(* CoDeSys 2.3 library: TcIoFunctions.lib *)
(* Libraries: STANDARD.LIB 5.6.98 17:03:02, TcBase.lib 14.5.09 17:14:08, TcSystem.lib 9.3.10 16:21:30, TcUtilities.lib*24.1.11 11:36:10 *)

(* Global variable list: Globale_Variablen *)
VAR_GLOBAL
END_VAR
VAR_GLOBAL CONSTANT
	ERROR_ASI_COMM_ERROR				:BYTE:=1;
	ERROR_ASI_SLAVEADDRESS				:BYTE:=2;
	ERROR_ASI_SLAVE_NOT_IN_LAS			:BYTE:=11;
	ERROR_ASI_TOGGLE_ERROR				:BYTE:=12;
	EEROR_ASI_DATAEXCHANGE_NOT_SET		:BYTE:=13;

	(* DPV1 via ProfiNET *)
	iMAX_DPV1_SIZE 			: INT := 240;
	iMAX_DPV1_PARAMS 		: INT := 39;

	(* DPV1 via ProfiNET *)
	iMAX_PNET_SIZE 	 		: INT := 32;
	iMAX_PNET_PARAMS 		: INT := 1;

	iMAX_DPV1_SIZE_PNET_REQ	: INT := 260;
	iMAX_DPV1_SIZE_PNET_RES	: INT := 240;

	iMAX_DRIVES_PER_CU		: INT := 15;
	iMAX_FAULTS_PER_DRIVE	: INT := 15;
END_VAR

(* Data type *)
TYPE ControlActiveConfiguration_t :
STRUCT
	HighSwitchCode : BYTE;
	LowSwitchCode : BYTE;
	High1 : BYTE;
	Low1 : BYTE;
	HighDeviceNo : BYTE;
	LowDeviceNo : BYTE;
END_STRUCT
END_TYPE

(* Data type *)
TYPE E_BatteryStatus :
(
	BatteryUnknownStatus, (*The battery status is unknown.*)
	BatteryOk, (*The batteries are OK.*)
	BatteryReplace (*The batteries need to be replaced.*)
);
END_TYPE

(* Data type *)
TYPE E_IOACCESSTYPE :
(
	eIOAccess_Default, 		(* normal memcpy function can be used to copy the data*)
	eIOAccess_Byte,			(* only byte access is allowed,  each byte of the data must be copied individually in a for loop *)
	eIOAccess_WordSwap	(* only aligned word access is allowed. High byte and low byte must be swapped *)
);
END_TYPE

(* Data type *)
TYPE E_PD_Datatype : (
	ePD_UNDEFINED		:=  0,
	ePD_BOOL			:=  1, (* 0/1 (not impl.) *)
	ePD_INT08			:=  2, (* -128 .. 127 *)
	ePD_INT16			:=  3, (* -32768 .. 32767 *)
	ePD_INT32			:=  4, (* -2147483648 .. 2147483647 *)
	ePD_UINT08			:=  5, (* 0 .. 255 *)
	ePD_UINT16			:=  6, (* 0 .. 65535 *)
	ePD_UINT32			:=  7, (* 0 .. 4294967295 *)
	ePD_FLOAT			:=  8, (* IEEE 754 *)
	ePD_VSTRING			:=  9, (* ISO/IEC 646, variable length *)
	ePD_OCTSTRING		:= 10, (* bytearray, variable length *)
	ePD_TIMEOFDAY_WDI	:= 12, (* 6 Bytes:
									4 bytes ms 
									+ 2 bytes day since 1.1.1984 *)
	ePD_TIMEDIFF		:= 13, (* 4|6 Bytes:
									4 bytes ms 
									+ optional 2 bytes days *)
	ePD_N2_16BIT		:= 33,
	ePD_N4_32BIT		:= 34,
	ePD_V2_BITSEQ		:= 35,
	ePD_L2_NIBBLE		:= 36,
	ePD_R2_RECIP_TC		:= 37,
	ePD_T2_TC_16BIT		:= 38,
	ePD_T2_TC_32BIT		:= 39,
	ePD_D2_TC			:= 40,
	ePD_E2_FIXPT_16		:= 41,
	ePD_C2_FIXPT_32		:= 42,
	ePD_X2_NV_16		:= 43,
	ePD_X4_NV_32		:= 44,
	ePD_DATE			:= 50, (* 7 Bytes:
									2 bytes ms
									+ 2 bits (res.), 6 bits (minutes) 
									+ 1 bit (0: StdTime/1: DaylightSavingTime), 2 bits (res.), 5 bits (hours) 
									+ 3 bits (DayOfWeek), 5 bits (DayOfMonth) 
									+ 2 bits (res.), 6 bits (month) 
									+ 1 bit (res.), 7 bits (year) *)
	ePD_TIMEOFDAY_NODI	:= 52, (* 0 .. 268435455 ms *)
	ePD_TIMEDIFF_WDI	:= 53, (* 6 Bytes:
									4 bytes ms 
									+ 2 bytes days *)
	ePD_TIMEDIFF_NODI	:= 54, (* 0 .. 4294967295 ms *)

	ePD_ZERO 			:= 64,
	ePD_BYTE 			:= 65,
	ePD_WORD 			:= 66,
	ePD_DWORD			:= 67,
	ePD_ERROR 			:= 68
);
END_TYPE

(* Data type *)
TYPE E_PD_Dpv1Error : (
	ePD_Err_ParamNumber 			:= 0,
	ePD_Err_ParamReadOnly			:= 1,
	ePD_Err_ValueOutOfRange			:= 2,
	ePD_Err_InvalidSubIndex			:= 3,
	ePD_Err_NoArray					:= 4,
	ePD_Err_WrongDataType			:= 5,
	ePD_Err_OnlyResetPermitted		:= 6,
	ePD_Err_DescNotChangable		:= 7,
	ePD_Err_DescNotFound			:= 9,
	ePD_Err_NoPermissionToChange	:= 11,
	ePD_Err_NoTextArray				:= 15,
	ePD_Err_JobNotExecutable		:= 17,
	ePD_Err_ValueInvalid			:= 20,
	ePD_Err_ResponseToLong			:= 21,
	ePD_Err_ParamAddrInvalid		:= 22,
	ePD_Err_FormatInvalid			:= 23,
	ePD_Err_NumOfValuesInvalid		:= 24,
	ePD_Err_DriveObjNotExisting		:= 25,
	ePD_Err_ParamDeactivated		:= 101,
	ePD_Err_ParamNoWrIfEnabled		:= 107,
	ePD_Err_ParamInvalidUnit		:= 108,
	ePD_Err_ParamNoWrIfNotInitFbk	:= 109,
	ePD_Err_ParamWrIfInitMtr		:= 110,
	ePD_Err_ParamWrIfInitDrv		:= 111,
	ePD_Err_ParamWrIfFastInit		:= 112,
	ePD_Err_ParamWrIfReady			:= 113,
	ePD_Err_ParamWrIfInitParamReset	:= 114,
	ePD_Err_ParamWrIfInitSafety		:= 115,
	ePD_Err_ParamWrIfInitTechApp	:= 116,
	ePD_Err_ParamWrIfInit			:= 117,
	ePD_Err_ParamWrIfInitDwnLd		:= 118,
	ePD_Err_ParamNoWrtIfDwnLd		:= 119,
	ePD_Err_ParamWrIfInitDrvCfg		:= 120,
	ePD_Err_ParamWrIfInitSetDrvType	:= 121,
	ePD_Err_ParamWrIfInitDatasetCfg	:= 122,
	ePD_Err_ParamWrIfInitDevCfg		:= 123,
	ePD_Err_ParamWrIfInitDevDwnLd	:= 124,
	ePD_Err_ParamWrIfInitDevPrmReset:= 125,
	ePD_Err_ParamWrIfInitDevReady	:= 126,
	ePD_Err_ParamWrIfInitDevice		:= 127,
	ePD_Err_ParamNoWriteIfDwnLd		:= 129,
	ePD_Err_CtrlTakeOverBlocked		:= 130,
	ePD_Err_ParamBicoSetInvalid		:= 131,
	ePD_Err_ParamChangeBlocked		:= 132,
	ePD_Err_ParamNoAccessDefined	:= 133,
	ePD_Err_BelowDefinedMinimum		:= 200,
	ePD_Err_AboveDefinedMaximum		:= 201,
	ePD_Err_WriteNotPermitted		:= 204
);
END_TYPE

(* Data type *)
TYPE E_PD_DriveType : (
	ePD_DRVTYPE_UNKNOWN 	:= 0,
	ePD_SINAMICS_S 			:= 1,
	ePD_SINAMICS_G 			:= 2,
	ePD_SINAMICS_I 			:= 3,
	ePD_SINAMICS_CX32 		:= 4,
	ePD_SINAMICS_GM 		:= 5,
	ePD_SINAMICS_GL 		:= 7,
	ePD_ACTLINEMOD 			:= 10,
	ePD_SERVO 				:= 11,
	ePD_VECTOR 				:= 12,
	ePD_VECTOR_VM 			:= 13,
	ePD_VECTOR_GL 			:= 14,
	ePD_SMARTLINEMOD 		:= 20,
	ePD_BASICLINEMOD 		:= 30,
	ePD_ACTIVELINEMOD_MV 	:= 40,
	ePD_BASICLINEMOD_MV 	:= 41,
	ePD_TB30 				:= 100,
	ePD_DMC 				:= 150,
	ePD_TM31 				:= 200,
	ePD_TM41 				:= 201,
	ePD_TM17_HIGHFEATURE 	:= 202,
	ePD_TM15 				:= 203,
	ePD_TM15_SINAMICS 		:= 204,
	ePD_CU_LINK 			:= 254
);
END_TYPE

(* Data type *)
TYPE E_PD_SaveType : (
	E_PD_SaveInactive 			:= 0,
	E_PD_SaveNonVolatilePWRON	:= 1,
	E_PD_SaveNonVolatileP967_10	:= 10,
	E_PD_SaveNonVolatileP967_11	:= 11,
	E_PD_SaveNonVolatileP967_12	:= 12,
	E_PD_SaveNonVolatile_20		:= 20,
	E_PD_SaveNonVolatile_21		:= 21,
	E_PD_SaveNonVolatile_22		:= 22,
	E_PD_SaveNonVolatile_23		:= 23,
	E_PD_SaveNonVolatile_24		:= 24,
	E_PD_SaveNonVolatile_25		:= 25,
	E_PD_SaveNonVolatile_26		:= 26,
	E_PD_SaveVolatileP967_1011	:= 1011,
	E_PD_SaveVolatileP967_1012	:= 1012,
	E_PD_SaveVolatileP967_1013	:= 1013
);
END_TYPE

(* Data type *)
TYPE E_PD_State : (
	ePD_IDLE 			:= 0,
	ePD_InitialRead 	:= 1,
	ePD_InitialWrite 	:= 2,
	ePD_ReadParam 		:= 3,
	ePD_WriteParam 		:= 4,
	ePD_ReadDiagInfo 	:= 5,
	ePD_QuitErrorCU 	:= 6,
	ePD_ResetDrive 		:= 7,
	ePD_SaveParamCU 	:= 8,
	ePD_SaveParamDrive 	:= 9,
	ePD_ClearErrorCU 	:= 10,
	ePD_ClearErrorDrive	:= 11,
	ePD_QuitErrorDrive 	:= 12
);
END_TYPE

(* Data type *)
TYPE E_SercosAttribLen : (
	eLEN_2BYTE	:= 1,
	eLEN_4BYTE	:= 2,
	eLEN_8BYTE	:= 3,
	eLEN_V1BYTE	:= 4,
	eLEN_V2BYTE	:= 5,
	eLEN_V4BYTE	:= 6,
	eLEN_V8BYTE	:= 7
);
END_TYPE

(* Data type *)
TYPE E_SercosAttribType : (
	eType_BIN		:= 0,
	eType_UNSIGNED	:= 1,
	eType_SIGNED	:= 2,
	eType_HEX		:= 3,
	eType_ASCII		:= 4,
	eType_ID		:= 5,
	eType_FLOAT		:= 6
);
END_TYPE

(* Data type *)
TYPE E_SercosBackupState  : (
	eBkup_IDLE 						:=  0,
	eBkup_READ_IDNLIST_INI 			:=  1,
	eBkup_READ_IDNLIST_ACT 			:=  2,
	eBkup_FILEOPEN					:=  3,
	eBkup_FILECLOSE					:=  4,
	eBkup_CHECK_CRC_ACT 			:=  5,
	eBkup_UPDT_CRC_INI				:=  6,
	eBkup_UPDT_CRC_ACT 				:=  7,

	eBkup_BACKUP_WRITE_FILEHEADER 	:= 10,
	eBkup_BACKUP_PARAM_INI 			:= 11,
	eBkup_BACKUP_PARAM_ACT 			:= 12,
	eBkup_BACKUP_WRITE_HEADER 		:= 14,
	eBkup_BACKUP_WRITE_DATA 		:= 15,

	eBkup_RESTORE_READ_FILEHEADER 	:= 20,
	eBkup_RESTORE_READ_HEADER		:= 21,
	eBkup_RESTORE_READ_DATA 		:= 22,
	eBkup_RESTORE_PARAM_INI			:= 23,
	eBkup_RESTORE_PARAM_ACT			:= 24
);
END_TYPE

(* Data type *)
TYPE E_SercosParamDataType : (
	eDT_LIST	:= 0,
	eDT_INT,
	eDT_UINT,
	eDT_WORD,
	eDT_DINT,
	eDT_UDINT,
	eDT_DWORD,
	eDT_REAL,
	eDT_LREAL
);
END_TYPE

(* Data type *)
TYPE E_UpsCommStatus :
(
	UpsCommUnknownStatus,
	UpsCommOk, (*The communication path to the UPS is OK.*)
	UpsCommFailed (*The communication path to the UPS has failed.*)
);
END_TYPE

(* Data type *)
TYPE E_UpsPowerStatus :
(
	PowerUnknownStatus, (*The status of power is unknown.*)
	PowerOnLine, (* Power is OK.*)
	PowerOnBattery (*A power failure has occurred.*)
);
END_TYPE

(* Data type *)
TYPE FC310X_DIAG_DATA :
STRUCT
	ReceiveErrorCounter: WORD;
	RepeatCounter: ARRAY[0..8] OF WORD;
	NoAnswerCounter: DWORD;
	LastDpv1Error: ARRAY[0..3] OF BYTE;
	Reserved: ARRAY[0..3] OF BYTE;
	DP_Diag_Stationstatus_1: BYTE;
	DP_Diag_Stationstatus_2: BYTE;
	DP_Diag_Stationstatus_3: BYTE;
	DP_Diag_MasterAdd: BYTE;
	DP_Diag_IdentNumberHi: BYTE;
	DP_Diag_IdentNumberLo: BYTE;
	DP_Diag_ExtDiagData: ARRAY[0..237] OF BYTE;
END_STRUCT
END_TYPE

(* Data type *)
TYPE FC510X_DIAG_DATA :
STRUCT
	flags: WORD;
	pdoReceived:WORD;
	pdoFault: WORD;
	startUpFault: BYTE;
	sdoFault: BYTE;
	index: WORD;
	subindex: BYTE;
	dummy2: BYTE;
	errorClass: BYTE;
	errorCode: BYTE;
	additionalCode: WORD;
	readValue: DWORD;
	expectedValue: DWORD;
	noOfEmergencies: WORD;
	emergency: ARRAY[0..9,0..7] OF BYTE;
END_STRUCT
END_TYPE

(* Data type *)
TYPE GetErrorInfo_t :
STRUCT
	HighResult : BYTE;
	LowResult : BYTE;
	HighEntryCount : BYTE;
	LowEntryCount : BYTE;
	HighErrorCode : BYTE;
	LowErrorCode : BYTE;
	HighAddErrInfo : BYTE;
	LowAddErrInfo : BYTE;
END_STRUCT
END_TYPE

(* Data type *)
TYPE HLword_t :
STRUCT
	High : BYTE;
	Low : BYTE;
END_STRUCT
END_TYPE

(* Data type *)
TYPE IODEVICETYPES :
(
	IODEVICETYPE_UNKNOWN			:= 0,
	IODEVICETYPE_C1220				:= 1,			(* Beckhoff Lightbus-Master*)
	IODEVICETYPE_C1200				:= 2,			(* Beckhoff Lightbus-Master*)
	IODEVICETYPE_SPC3				:= 3,			(* ProfiBus Slave (Siemens)*)
	IODEVICETYPE_CIF30DPM			:= 4,			(* ISA ProfiBus-Master 2 kByte (Hilscher)*)
	IODEVICETYPE_CIF40IBSM			:= 5,			(* ISA Interbus-S-Master 2 kByte (Hilscher)*)
	IODEVICETYPE_BKHFPC			:= 6,			(* Beckhoff PC C2001*)
	IODEVICETYPE_CP5412A2			:= 7,			(* ProfiBus-Master (Siemens)*)
	IODEVICETYPE_SERCANSISA		:= 8,			(* Sercos Master (Indramat)*)
	IODEVICETYPE_LPTPORT			:= 9,			(* Lpt Port*)
	IODEVICETYPE_DPRAM				:= 10,		(* Generic DPRAM*)
	IODEVICETYPE_COMPORT			:= 11,		(* COM Port*)
	IODEVICETYPE_CIF30CAN			:= 12,		(* ISA CANopen-Master (Hilscher)*)
	IODEVICETYPE_CIF30PB			:= 13,		(* ISA ProfiBus-Master 8 kByte (Hilscher)*)
	IODEVICETYPE_BKHFCP2030		:= 14,		(* Beckhoff CP2030 (Pannel-Link)*)
	IODEVICETYPE_IBSSCIT				:= 15,		(* ISA Interbus-S-Master (Phoenix)*)
	IODEVICETYPE_CIF30IBM			:= 16,		(* ISA Interbus-S-Master (Hilscher)*)
	IODEVICETYPE_CIF30DNM			:= 17,		(* ISA DeviceNet-Master (Hilscher)*)
	IODEVICETYPE_FCXXXX				:= 18,		(* Beckhoff-Filedbus card *)
	IODEVICETYPE_CIF50PB			:= 19,		(* PCI ProfiBus-Master 8 kByte (Hilscher)*)
	IODEVICETYPE_CIF50IBM			:= 20,		(* PCI Interbus-S-Master (Hilscher)*)
	IODEVICETYPE_CIF50DNM			:= 21,		(* PCI DeviceNet-Master (Hilscher)*)
	IODEVICETYPE_CIF50CAN			:= 22,		(* PCI CANopen-Master (Hilscher)*)
	IODEVICETYPE_CIF60PB			:= 23,		(* PCMCIA ProfiBus-Master (Hilscher)*)
	IODEVICETYPE_CIF60DNM			:= 24,		(* PCMCIA DeviceNet-Master (Hilscher)*)
	IODEVICETYPE_CIF60CAN			:= 25,		(* PCMCIA CANopen-Master (Hilscher)*)
	IODEVICETYPE_CIF104DP			:= 26,		(* PC104 ProfiBus-Master 2 kByte (Hilscher)*)
	IODEVICETYPE_C104PB				:= 27,		(* PC104 ProfiBus-Master 8 kByte (Hilscher)*)
	IODEVICETYPE_C104IBM			:= 28,		(* PC104 Interbus-S-Master 2 kByte (Hilscher)*)
	IODEVICETYPE_C104CAN			:= 29,		(* PC104 CANopen-Master (Hilscher)*)
	IODEVICETYPE_C104DNM			:= 30,		(* PC104 DeviceNet-Master (Hilscher)*)
	IODEVICETYPE_BKHFCP9030		:= 31,		(* Beckhoff CP9030 (Pannel-Link with UPS)*)
	IODEVICETYPE_SMB					:= 32,		(* Motherboard System Management Bus*)
	IODEVICETYPE_PBMON				:= 33,		(* Beckhoff-PROFIBUS-Monitor*)
	IODEVICETYPE_CP5613				:= 34,		(* PCI ProfiBus-Master (Siemens)*)
	IODEVICETYPE_CIF60IBM			:= 35,		(* PCMCIA Interbus-S-Master (Hilscher)*)
	IODEVICETYPE_FC200X				:= 36,		(* Beckhoff-Lightbus-I/II-PCI-Karte*)
	IODEVICETYPE_FC3100_OLD		:= 37,		(* obsolete: dont use*)
	IODEVICETYPE_FC3100				:= 38,		(* Beckhoff-Profibus-PCI*)
	IODEVICETYPE_FC5100				:= 39,		(* Beckhoff-CanOpen-PCI*)
	IODEVICETYPE_FC5200				:= 41,		(* Beckhoff-DeviceNet-PCI*)

	IODEVICETYPE_BKHFNCBP			:= 43,		(* Beckhoff NC back plane*)
	IODEVICETYPE_SERCANSPCI		:= 44,		(* Sercos Master (SICAN/IAM PCI)*)
	IODEVICETYPE_ETHERNET			:= 45,		(* Virtual Ethernet Device*)
	IODEVICETYPE_SERCONPCI		:= 46,		(* Sercon 410B or 816 Chip Master or Slave (PCI)*)
	IODEVICETYPE_IBSSCRIRTLK		:= 47,		(* ISA Interbus-S-Master with Slave-Module LWL Basis (Phoenix)*)
	IODEVICETYPE_FC7500				:= 48,		(* Beckhoff-SERCOS-PCI*)
	IODEVICETYPE_CIF30IBS			:= 49,		(* ISA Interbus-S-Slave (Hilscher)*)
	IODEVICETYPE_CIF50IBS			:= 50,		(* PCI Interbus-S-Slave (Hilscher)*)
	IODEVICETYPE_C104IBS			:= 51,		(* PC104 Interbus-S-Slave (Hilscher)*)
	IODEVICETYPE_BKHFCP9040		:= 52,		(* Beckhoff CP9040 (CP-PC) *)
	IODEVICETYPE_BKHFAH2000		:= 53,		(* Beckhoff AH2000 (Hydr. Backplane) *)
	IODEVICETYPE_BKHFCP9035		:= 54,		(* Beckhoff CP9035 (PCI, Pannel-Link with UPS) *)
	IODEVICETYPE_AH2000MC			:= 55,		(* Beckhoff-AH2000 with Profibus-MC *)
	IODEVICETYPE_FC3100MON		:= 56,		(* Beckhoff-Profibus-Monitor-PCI *)
	IODEVICETYPE_USB					:= 57,		(* Virtual USB Device *)
	IODEVICETYPE_FC5100MON		:= 58,		(* Beckhoff-CANopen-Monitor-PCI *)
	IODEVICETYPE_FC5200MON		:= 59,		(* Beckhoff-DeviceNet-Monitor-PCI *)
	IODEVICETYPE_FC3100SLV			:= 60,		(* Beckhoff-Profibus-PCI Slave *)
	IODEVICETYPE_FC5100SLV			:= 61,		(* Beckhoff-CanOpen-PCI Slave *)
	IODEVICETYPE_FC5200SLV			:= 62,		(* Beckhoff-DeviceNet-PCI Slave *)
	IODEVICETYPE_IBSSCITPCI			:= 63,		(* PCI Interbus-S-Master (Phoenix) *)
	IODEVICETYPE_IBSSCRIRTLKPCI	:= 64,		(* PCI Interbus-S-Master with slave module  LWL Basis (Phoenix) *)
	(* 11 November 2002 *)
	IODEVICETYPE_CX1100_BK		:= 65,		(* Beckhoff-CX1100 terminal bus power supply *)
	IODEVICETYPE_ENETRTMP			:= 66,		(* Ethernet real time miniport *)
	IODEVICETYPE_CX1500_M200		:= 67,		(* PC104 Lightbus-Master *)
	IODEVICETYPE_CX1500_B200		:= 68,		(* PC104 Lightbus-Slave *)
	IODEVICETYPE_CX1500_M310		:= 69,		(* PC104 ProfiBus-Master *)
	IODEVICETYPE_CX1500_B310		:= 70,		(* PC104 ProfiBus-Slave *)
	IODEVICETYPE_CX1500_M510		:= 71,		(* PC104 CANopen-Master *)
	IODEVICETYPE_CX1500_B510		:= 72,		(* PC104 CANopen-Slave *)
	IODEVICETYPE_CX1500_M520		:= 73,		(* PC104 DeviceNet-Master *)
	IODEVICETYPE_CX1500_B520		:= 74,		(* PC104 DeviceNet-Slave *)
	IODEVICETYPE_CX1500_M750		:= 75,		(* PC104 Sercos-Master *)
	IODEVICETYPE_CX1500_B750		:= 76,		(* PC104 Sercos-Slave *)
	IODEVICETYPE_BX_BK				:= 77,		(* BX terminal bus interface *)
	IODEVICETYPE_BX_M510			:= 78,		(* BX SSB-Master *)
	IODEVICETYPE_BX_B310			:= 79,		(* BX ProfiBus-Slave *)
	(* 29 August 2005 *)
	IODEVICETYPE_IBSSCRIRTPCI		:= 80,		(* PCI Interbus-S-Master with slave module copper basis (Phoenix) *)
	IODEVICETYPE_BX_B510			:= 81,		(* BX CANopen Slave *)
	IODEVICETYPE_BX_B520			:= 82,		(* BX DeviceNet Slave *)
	IODEVICETYPE_BC3150				:= 83,		(* BCxx50 ProfiBus Slave *)
	IODEVICETYPE_BC5150				:= 84,		(* BCxx50 CANopen Slave *)
	IODEVICETYPE_BC5250				:= 85,		(* BCxx50 DeviceNet Slave *)
	IODEVICETYPE_EL6731				:= 86,		(* Beckhoff Profibus-EtherCAT Terminal *)
	IODEVICETYPE_EL6751				:= 87,		(* Beckhoff CanOpen-EtherCAT Terminal *)
	IODEVICETYPE_EL6752				:= 88,		(* Beckhoff DeviceNet-EtherCAT Terminal *)
	IODEVICETYPE_COMPB				:= 89,		(* COM ProfiBus Master 8 kByte (Hilscher) *)
	IODEVICETYPE_COMIBM			:= 90,		(* COM Interbus-S Master (Hilscher) *)
	IODEVICETYPE_COMDNM			:= 91,		(* COM DeviceNet Master (Hilscher) *)
	IODEVICETYPE_COMCAN			:= 92,		(* COM CANopen Master (Hilscher) *)
	IODEVICETYPE_COMIBS				:= 93,		(* COM CANopen Slave (Hilscher) *)
	IODEVICETYPE_ETHERCAT			:= 94,		(* EtherCAT in direct mode *)
	IODEVICETYPE_PROFINETIOCONTROLLER := 95,	(* PROFINET Master *)
	IODEVICETYPE_PROFINETIODEVICE := 96,		(* PROFINET Slave *)
	IODEVICETYPE_EL6731SLV			:= 97,		(* Beckhoff Profibus Slave EtherCAT Terminal *)
	IODEVICETYPE_EL6751SLV			:= 98,		(* Beckhoff CanOpen Slave EtherCAT Terminal *)
	IODEVICETYPE_EL6752SLV			:= 99,		(* Beckhoff DeviceNet Slave EtherCAT Terminal *)
	IODEVICETYPE_C104PPB			:= 100,		(* PC104+ ProfiBus Master 8 kByte (Hilscher) *)
	IODEVICETYPE_C104PCAN			:= 101,		(* PC104+ CANopen Master (Hilscher) *)
	IODEVICETYPE_C104PDNM			:= 102,		(* PC104+ DeviceNet Master (Hilscher) *)
	IODEVICETYPE_BC8150				:= 103,		(* BCxx50 Serial Slave *)
	IODEVICETYPE_BX9000				:= 104,		(* BX9000 Ethernet Slave *)
	(* 27 April 2009 *)
	IODEVICETYPE_CX9000_BK		:= 105,	(* Beckhoff-CX9000 K-Bus Power Supply *)
	IODEVICETYPE_EL6601				:= 106,	(* Beckhoff-RT-Ethernet-EtherCAT-Terminal *)
	IODEVICETYPE_BC9050				:= 107,	(* BC9050 Ethernet Slave *)
	IODEVICETYPE_BC9120				:= 108,	(* BC9120 Ethernet Slave *)
	IODEVICETYPE_ENETADAPTER	:= 109,	(* Ethernet Miniport Adapter *)
	IODEVICETYPE_BC9020				:= 110,	(* BC9020 Ethernet Slave *)
	IODEVICETYPE_ETHERCATPROT	:= 111,	(* EtherCAT Protocol in direct mode *)
	IODEVICETYPE_ETHERNETNVPROT	:= 112,	(* *)
	IODEVICETYPE_ETHERNETPNMPROT	:= 113,	(* *)
	IODEVICETYPE_EL6720				:= 114,	(* Beckhoff-Lightbus-EtherCAT-Terminal *)
	IODEVICETYPE_ETHERNETPNSPROT	:= 115,	(* *)
	IODEVICETYPE_BKHFCP6608		:= 116,	(*	Beckhoff CP6608(IXP PC) *)
	IODEVICETYPE_PTP_IEEE1588		:= 117,  (* *)
	IODEVICETYPE_EL6631SLV			:= 118,	(* EL6631-0010 Profinet Slave terminal *)
	IODEVICETYPE_EL6631				:= 119,	(* EL6631 Profinet Master terminal *)
	IODEVICETYPE_CX5000_BK		:= 120,	(* Beckhoff-CX5100 K-Bus power supply *)
	IODEVICETYPE_PCIDEVICE			:= 121,	(* Generic PCI DPRAM (TCOM) *)
	IODEVICETYPE_ETHERNETUPDPROT 	:= 122,	(* UDP Protocol *)
	(* 13 August 2010 *)
	IODEVICETYPE_ETHERNETAUTOPROT := 123,	(* Automation Protocol *)
	IODEVICETYPE_CCAT				:= 124,	(* CCAT *)
	IODEVICETYPE_CPLINK3			:= 125,	(* Virtuelles USB Device (remote via CPLINK3) *)
	IODEVICETYPE_EL6632				:= 126,	(* EL6632 *)
	IODEVICETYPE_CCAT_PBM			:= 127,	(* CCAT Profibus Master *)
	IODEVICETYPE_CCAT_PBS			:= 128,	(* CCAT Profibus Slave *)
	IODEVICETYPE_CCAT_CNM			:= 129,	(* CCAT CANopen Master *)
	IODEVICETYPE_ETHERCATSLAVE	:= 130,	(* EtherCAT Slave *)
	IODEVICETYPE_BACNET			:= 131,	(* BACnet device *)
	IODEVICETYPE_CCAT_CNS			:= 132,	(* CCAT CANopen Slave *)
	IODEVICETYPE_ETHIP_SCANNER	:= 133,  (* ETHERNET IP  Master *)
	IODEVICETYPE_ETHIP_ADAPTER	:= 134,  (* ETHERNET IP  Slave *)

	(* reserved for new devices*)

	IODEVICETYPE_MAX							(**)
);
END_TYPE

(* Data type *)
TYPE ReadResult_t :
STRUCT
	High1 : BYTE;
	Low1 : BYTE;
	High2 : BYTE;
	Low2 : BYTE;
END_STRUCT
END_TYPE

(* Data type *)
TYPE ST_AdsTecSysData :
STRUCT
	bShiftKey		: BOOL; 	(* TRUE == Shift key pressed*)
	bRMouseKey		: BOOL; 	(* TRUE == Right mouse key pressed *)
	bHotKey			: BOOL;	(* TRUE == Hotkey pressed *)
	bTaskChaKey	: BOOL;	(* TRUE == Task change key pressed *)
	bABCKey		: BOOL;	(* TRUE == ABC soft keyboard key pressed*)
	bRsrv1			: BOOL;
	bRsrv2			: BOOL;
	bRsrv3			: BOOL;

	bMainFanErr		: BOOL; 	(* TRUE == Main fan error*)
	bCpuFanErr		: BOOL;	(* TRUE == CPU fan error*)
	bTempErr		: BOOL;	(* TRUE == Internal temperature error ( temp > 50°C)*)
	bBatteryErr		: BOOL;	(* TRUE == Battery error *)
	bRsrv4			: BOOL;
	bRsrv5			: BOOL;
	bRsrv6			: BOOL;
	bRsrv7			: BOOL;

	nMainNtcTemp	: SINT; 	(* Main NTC temperature (-127°C .. + 127°C) *)
	nExtNtcTemp		: SINT;	(* External NTC temperature (-127°C .. + 127°C) *)

	nRsrv8			: ARRAY[1..12] OF BYTE;
END_STRUCT
END_TYPE

(* Data type *)
TYPE ST_Dpv1Header :
STRUCT
	(* header *)
	iRequestRef 	: USINT;	(* 1..255;    0: reserved *)
	iRequestID 		: SINT;		(* 1: Read;   2: Write;     0x40..0x7F: manufacturer specific;   else: reserved *)
	iAxis			: USINT;	(* 0..255 *)
	iNumOfParams	: USINT;	(* 1..39;     else: reserved *)
END_STRUCT
END_TYPE

(* Data type *)
TYPE ST_Dpv1ParamAddr :
STRUCT
	(* parameter *)
	iAttribute			: USINT;	(* 0x10: Value;   0x20: Description;   0x30: Text (not impl.);   0x80..F0: manufaturer specific (not impl.);   else: reserved *)
	iNumOfElements		: USINT;	(* 1..117: number of array elements;    0: Special Function;   else: reserved *)
	iParameterNumber	: UINT;		(* 1..65535: parameter number;    0: reserved *)
	iSubIndex			: UINT;		(* 0..65535: subindex *)
END_STRUCT
END_TYPE

(* Data type *)
TYPE ST_Dpv1ParamAddrEx :
STRUCT
	(* parameter *)
	iAttribute			: USINT;	(* 0x10: Value;   0x20: Description;   0x30: Text;   0x80..F0: manufaturer specific;   else: reserved *)
	iNumOfElements		: USINT;	(* 1..234: number of elements;    0: Special Function;   else: reserved *)
	iParameterNumber	: UINT;		(* 1..65535: parameter number;    0: reserved *)
	iSubIndex			: UINT;		(* 0..65535: subindex *)
	iDataAddr			: UDINT;	(* address of buffer/address of plc variable *)
	iDataSize			: UDINT;	(* size of buffer/size of plc variable *)
	eFormat				: E_PD_Datatype;	(* 0x01..0x36: datatype;   0x40: ZERO;   0x41: BYTE;   0x42: WORD;   0x43: DWORD;   0x44: Error;   else reserved *)
	iNumOfValues		: UINT;		(* 0..234: number of values;   else: reserved *)
	iErrorValue			: UDINT;	(* DPV1 error value *)
	stError				: ST_PD_Dpv1Error; (* DPV1 error flag, DPV1 error enum *)
END_STRUCT
END_TYPE

(* Data type *)
TYPE ST_Dpv1ValueHeader :
STRUCT
	iFormat			: USINT;	(* 0x01..0x36: datatype;   0x40: ZERO;   0x41: BYTE;   0x42: WORD;   0x43: DWORD;   0x44: Error;   else reserved *)
	iNumOfValues	: USINT;	(* 0..234: number of values;   else: reserved *)
END_STRUCT
END_TYPE

(* Data type *)
TYPE ST_Dpv1ValueHeaderEx :
STRUCT
	eFormat			: E_PD_Datatype;	(* 0x01..0x36: datatype;   0x40: ZERO;   0x41: BYTE;   0x42: WORD;   0x43: DWORD;   0x44: Error;   else reserved *)
	iNumOfValues	: USINT;	(* 0..234: number of values;   else: reserved *)
	iOffset			: USINT;	(* Offset in the DPV1 response telegram *)
	iDataLen		: UINT;		(* data lenght *)
	strData			: STRING;	(* printed data *)
END_STRUCT
END_TYPE

(* Data type *)
TYPE ST_NovRamAddrInfo :
STRUCT
	pCardAddress	:	UDINT;
	iCardMemSize	:	UDINT;
END_STRUCT
END_TYPE

(* Data type *)
TYPE ST_NovRamAddrInfoEx :
STRUCT
	pCardAddress	:	UDINT;
	iCardMemSize	:	UDINT;
	eAccessType	:	E_IOACCESSTYPE;
END_STRUCT
END_TYPE

(* Data type *)
TYPE ST_Parameter_IN :
STRUCT
	iParameterStatus			:WORD;
	iParameterReadValue		:DWORD;

(*ParameterStatus
Byte-Offset	Bit-Offset		Bedeutung
	0			0-5		Status-Bits (wie bei bisherigen Klemmen)
	0			6		0: keine Diagnose, 1: Diagnose (wie bei bisherigen Klemmen)
	0			7		immer 0: keine Registerkommunikation
	1			0-3		Reserviert für Erweiterungen
	1			4		Toggle-Bit, um Auftrag zu quittieren (bei Cyclic wird das Bit 6 aus Byte 0 kopiert)
	1			5		Quittung (0: NoError, 1: Error)
	1			6		0: Cyclic, 1: Acyclic
	1			7		0: Parameterzugriff, 1: ADS
	2					Input-Daten (Cyclic), Parameterwert (Acyclic) oder Fehlernummer Bit 0-7
	3					Input-Daten (Cyclic), Parameterwert (Acyclic) oder Fehlernummer Bit 8-15
	4					Input-Daten (Cyclic), Parameterwert (Acyclic) oder Fehlernummer Bit 16-23
	5					Input-Daten (Cyclic), Parameterwert (Acyclic) oder Fehlernummer Bit 24-31

*)
END_STRUCT
END_TYPE

(* Data type *)
TYPE ST_Parameter_OUT :
STRUCT
	ParameterControl			:WORD;
	iParametervalue			:DWORD;

(*ParameterControl
Byte-Offset	Bit-Offset		Bedeutung
	0			0-5		Parameternummer Bit 0-5 (oder Parameter-Offset)
	0			6		Bei Acyclic: 0: Read, 1:Write, bei Cyclic (immer Read/Write) wird das Bit in die Inputdaten kopiert, um eine direkte Zuordnung zu haben (dann könnten die Cyclic-Daten auch geändert werden)
	0			7		0: Parameterzugriff, 1: Registerkommunikation
	1			0-5		Parameternummer Bit 6-11 (oder Parameter-Page)
	1			6		0: Cyclic, 1: Acyclic
	1			7		0: Parameterzugriff, 1: ADS
	2					Output-Daten (Cyclic) oder Parameterwert (Acyclic) Bit 0-7
	3					Output-Daten (Cyclic) oder Parameterwert (Acyclic) Bit 8-15
	4					Output-Daten (Cyclic) oder Parameterwert (Acyclic) Bit 16-23
	5					Output-Daten (Cyclic) oder Parameterwert (Acyclic) Bit 24-31

*)

END_STRUCT
END_TYPE

(* Data type *)
TYPE ST_ParameterBuffer :
STRUCT
	ParameterControl			:ARRAY[0..50] OF WORD;
	iParametervalue			:ARRAY[0..50] OF DWORD;
	iParameterStatus			:ARRAY[0..50] OF WORD;
	iParameterReadValue		:ARRAY[0..50] OF DWORD;
	icounterState				:INT;
	icounterControl			:INT;
END_STRUCT
END_TYPE

(* Data type *)
TYPE ST_PD_CUDriveInfo :
STRUCT
	iNumOfDriveObjects	: UINT;
	iReserved	: UINT;
	iIndex		: ARRAY [0..iMAX_DRIVES_PER_CU] OF UINT;			(* [0] is ControlUnit, [1..15] for the drives *)
	eType		: ARRAY [0..iMAX_DRIVES_PER_CU] OF E_PD_DriveType;	(* [0] is ControlUnit, [1..15] for the drives *)
	iFWVersion	: ARRAY [0..iMAX_DRIVES_PER_CU] OF UDINT;			(* [0] is ControlUnit, [1..15] for the drives *)
	iFWDateYear	: ARRAY [0..iMAX_DRIVES_PER_CU] OF UINT;			(* [0] is ControlUnit, [1..15] for the drives *)
	iFWDateDM	: ARRAY [0..iMAX_DRIVES_PER_CU] OF UINT;			(* [0] is ControlUnit, [1..15] for the drives *)
	iPbTelType	: ARRAY [0..iMAX_DRIVES_PER_CU] OF UINT;			(* [0] is ControlUnit, [1..15] for the drives *)
END_STRUCT
END_TYPE

(* Data type *)
TYPE ST_PD_DOIdentification :
STRUCT
	iCompany				: UINT;				(* 42 = Siemens *)
	eType					: E_PD_DriveType;	(* drive object type, e.g. ePD_SINAMICS_S, ePD_SERVO, ... *)
	iFWVersion				: UINT;				(* 102 --> v01.02, hotfix see below *)
	iFWDateYear				: UINT;				(* 2003 --> year 2003 *)
	iFWDateDayMonth			: UINT;				(* 1401 --> 14.01. *)
	iProfiDrvTypeClass		: UINT;
	iProfiDrvSubTypeClass	: UINT;
	iReserved				: ARRAY [7..9] OF UINT;
	iFWVersionPatchVersion	: UINT;				(* 600 --> FW v01.02.06.00, hotfix see below *)
END_STRUCT
END_TYPE

(* Data type *)
TYPE ST_PD_Dpv1Error :
STRUCT
	bError		: BOOL;
	eErrorId	: E_PD_Dpv1Error;
END_STRUCT
END_TYPE

(* Data type *)
TYPE ST_PD_DriveDiag :
STRUCT
	iNumOfFaultsTotal		: UINT;
	iNumOfFaultsSinceReset	: UINT;
	iNumOfWarnsTotal		: UINT;
	iStateWordErrorWarning	: UINT;
	iErrorCode	: ARRAY [0..iMAX_FAULTS_PER_DRIVE] OF UINT;			(* [0] is ControlUnit, [1..15] for the drives *)
	iErrorArgI	: ARRAY [0..iMAX_FAULTS_PER_DRIVE] OF UDINT;		(* [0] is ControlUnit, [1..15] for the drives *)
	fErrorArgF	: ARRAY [0..iMAX_FAULTS_PER_DRIVE] OF REAL;			(* [0] is ControlUnit, [1..15] for the drives *)
	iWarnCode	: ARRAY [0..iMAX_FAULTS_PER_DRIVE] OF UINT;			(* [0] is ControlUnit, [1..15] for the drives *)
	iWarnArgI	: ARRAY [0..iMAX_FAULTS_PER_DRIVE] OF UDINT;		(* [0] is ControlUnit, [1..15] for the drives *)
	fWarnArgF	: ARRAY [0..iMAX_FAULTS_PER_DRIVE] OF REAL;			(* [0] is ControlUnit, [1..15] for the drives *)
END_STRUCT
END_TYPE

(* Data type *)
TYPE ST_PNET_CCDSTS :
STRUCT
	iCycleCounter	: UINT;
	iDataState		: USINT;
	iTransferState	: USINT;
END_STRUCT
END_TYPE

(* Data type *)
TYPE ST_PNIOConfigRecord :
STRUCT
	iRW				: UINT; (* 0: Read, 1: Write *)
	iNumOfAR		: UINT;
	iAPI			: UDINT;
	iSlot			: UINT;
	iSubSlot		: UINT;
	stPNIORecord	: ST_PNIORecord;
END_STRUCT
END_TYPE

(* Data type *)
TYPE ST_PNIORecord :
STRUCT
	iIndex 		: UINT;
	iLength 	: UINT; (* 0 for READ *)
	iTransfSeq	: UINT;
	iAligned 	: UINT;
END_STRUCT
END_TYPE

(* Data type *)
TYPE ST_PNIOState :
STRUCT
	bInDataExchange	: BOOL; (* bit 0 *)
	bApplRunning	: BOOL; (* bit 2 *)
	bDiagIndicator	: BOOL; (* bit 3 *)
END_STRUCT
END_TYPE

(* Data type *)
TYPE ST_PZD_IN :
STRUCT
	wSTW		:WORD;
	wHIW		:WORD;
	PZD3		:WORD;
	PZD4		:WORD;
	PZD5		:WORD;
	PZD6		:WORD;

END_STRUCT
END_TYPE

(* Data type *)
TYPE ST_PZD_OUT :
STRUCT
	wCtrlW			:WORD;
	PZD2			:WORD;
	PZD3			:WORD;
	PZD4			:WORD;
	PZD5			:WORD;
	PZD6			:WORD;
END_STRUCT
END_TYPE

(* Data type *)
TYPE ST_SercosFileHeader :
STRUCT
	nVersion	 : UDINT;
	nListType	 : UDINT;
	cbCommentLen : UDINT;
	sComment	 : T_MaxString;
END_STRUCT
END_TYPE

(* Data type *)
TYPE ST_SercosParamAttrib :
STRUCT
	nFactor			: UINT;					(* bits  0..15 *)
	eLength			: E_SercosAttribLen;	(* bits 16..18 *)
	bCommand		: BOOL;					(* bit  19     *)
	eType			: E_SercosAttribType;	(* bits 20..22 *)
	bReserved1		: BOOL;					(* bit  23     *)
	nComma			: USINT;				(* bits 24..27 *)
	bWriteProtCP2	: BOOL;					(* bit  28     *)
	bWriteProtCP3	: BOOL;					(* bit  29     *)
	bWriteProtCP4	: BOOL;					(* bit  30     *)
	bReserved2		: BOOL;					(* bit  31     *)
END_STRUCT
END_TYPE

(* Data type *)
TYPE ST_SercosParamData :
STRUCT
	nAttrib		: DWORD;
	sAttrib		: ST_SercosParamAttrib;
	eDataType	: E_SercosParamDataType;

	cbValLenAct	: UINT;
	cbValLenMax	: UINT;
	arrData		: ARRAY [0..65535] OF BYTE;

	sName		: ST_SercosString;
	sUnit		: ST_SercosString;

	nMinArr		: ARRAY[0..7] OF BYTE;
	nMaxArr		: ARRAY[0..7] OF BYTE;
END_STRUCT
END_TYPE

(* Data type *)
TYPE ST_SercosParamErrList :
STRUCT
	iActCount	: UINT;
	iMaxCount	: UINT;
	iList		: ARRAY [0..2047] OF UINT;
	iError		: ARRAY [0..2047] OF UDINT;
END_STRUCT
END_TYPE

(* Data type *)
TYPE ST_SercosParamHeader :
STRUCT
	nIDN		: UINT;
	cbSize		: UINT;
	nAttrib		: DWORD;
END_STRUCT
END_TYPE

(* Data type *)
TYPE ST_SercosParamList :
STRUCT
	iActCount	: UINT;
	iMaxCount	: UINT;
	iList		: ARRAY [0..2047] OF UINT;
END_STRUCT
END_TYPE

(* Data type *)
TYPE ST_SercosString :
STRUCT
	iActSize	: UINT;
	iMaxSize	: UINT;
	sString		: STRING(255);
END_STRUCT
END_TYPE

(* Data type *)
TYPE ST_UPSStatus :
STRUCT
	Vendor					: STRING;
	Model					: STRING;
	FirmwareRev				: STRING; (*Reports the UPS firmware revision as a displayable string. *)
	SerialNumber				: STRING; (*Reports the UPS serial number as a displayable string.*)
	BatteryLifePercent 		: DWORD; (* The percent of battery capacity remaining in the UPS, represented as a value in the range of 0 through 100. *)
	BatteryLifeTime 			: DWORD; (*The amount of remaining UPS run time, in minutes.*)
	eBatteryStatus			: E_BatteryStatus; (*The current status of the UPS batteries. *)
	eCommStatus			: E_UpsCommStatus; (*The status of the communication path to the UPS. *)
	ePowerStatus				: E_UpsPowerStatus; (* Reports the status of utility-supplied power into the UPS. *)
	nPowerFailCnt			: DWORD; (* Power fail counter *)
	dwChargeFlags			: DWORD; (*	Reserved for future use.
		Battery charge status flags. This member can be one or more of the following values.
		0:	Unknown status
		1: 	High
		2: 	Low
		4: 	Critical
		8:	Charging
		128:	No battery
	 *)
END_STRUCT
END_TYPE

(* POU F_ByteSwap, ST *)
FUNCTION F_ByteSwap : INT
(*****************************************************************************************************************
	DESCRIPTION:	This FUNCTION swaps bytes of lager datatypes (Intel Format <-> Motorola Format)

	CHANGE LOG:
	BY		DATE		DESCRIPTION OF CHANGE
	ICh		2006/07/12	bugfix for arrays of known type elements
	ICh		2006/07/05	First Version

******************************************************************************************************************)
VAR_INPUT
	pSrcAdr			: POINTER TO BYTE := 0;
	pDstAdr			: POINTER TO BYTE := 0;
	iSize			: USINT := 0;
	eType			: E_PD_Datatype := ePD_UNDEFINED;
END_VAR
VAR
	iByte			: BYTE;
	iIndex			: USINT;
	iTypeSize		: USINT;
	bEven			: BOOL;
	bOdd			: BOOL;
	iRepeats		: INT;

	pSrcAdrPtr		: POINTER TO BYTE;
	pSrcAdrPtrOrg	: POINTER TO BYTE;
	pDstAdrPtr		: POINTER TO BYTE;
	pDstAdrPtrOrg	: POINTER TO BYTE;
END_VAR
IF (pSrcAdr = 0) OR (pDstAdr = 0) OR (iSize = 0) THEN
	(* error *)
	pSrcAdrPtr := pSrcAdr;
	pDstAdrPtr := pDstAdr;

	F_ByteSwap := -1;

ELSIF pSrcAdr = pDstAdr THEN
	(* swap directly in the srcData *)
	pSrcAdrPtr	:= pSrcAdr;
	iTypeSize	:= F_GetPDTypeSize(eType);
	iRepeats	:= 0;
	bEven		:= FALSE;
	bOdd		:= FALSE;

	IF iTypeSize <> 0 THEN
		IF (iSize = iTypeSize) THEN
			(* single element *)
			pDstAdrPtr	:= pDstAdr + USINT_TO_DWORD(iSize - 1);
		ELSIF iSize > iTypeSize THEN
			pDstAdrPtr	:= pDstAdr + USINT_TO_DWORD(iTypeSize - 1);
			iRepeats	:= iSize / iTypeSize - 1;

			IF iRepeats < 0 THEN
				iRepeats := 0;
			END_IF

			IF (iSize MOD iTypeSize) = 0 THEN
				(* array, n-times element size matches block size *)
				bEven := TRUE;
			ELSE
				(* array, n-times element size does not match block size *)
				bOdd := TRUE;
			END_IF
		ELSE
			(* treat as single element *)
			pDstAdrPtr	:= pDstAdr + USINT_TO_DWORD(iSize - 1);
			iTypeSize	:= iSize;
		END_IF
	ELSE
		(* treat as single element *)
		pDstAdrPtr	:= pDstAdr + USINT_TO_DWORD(iSize - 1);
		iTypeSize	:= iSize;
	END_IF

	pSrcAdrPtrOrg := pSrcAdrPtr;
	pDstAdrPtrOrg := pDstAdrPtr;

	(* execute at least once *)
	REPEAT
		FOR iIndex := 0 TO iSize-1 DO
			iByte 		:= pDstAdrPtr^;
			pDstAdrPtr^	:= pSrcAdrPtr^;
			pSrcAdrPtr^	:= iByte;
			pSrcAdrPtr	:= pSrcAdrPtr + DWORD#1;
			pDstAdrPtr	:= pDstAdrPtr - DWORD#1;
			IF pDstAdrPtr <= pSrcAdrPtr THEN
				EXIT;
			END_IF
		END_FOR

		IF bEven OR bOdd THEN
			pSrcAdrPtr		:= pSrcAdrPtrOrg + USINT_TO_DWORD(iTypeSize);
			pSrcAdrPtrOrg	:= pSrcAdrPtr;
			pDstAdrPtr		:= pDstAdrPtrOrg + USINT_TO_DWORD(iTypeSize);
			pDstAdrPtrOrg	:= pDstAdrPtr;
		END_IF

		iRepeats := iRepeats - 1;
	UNTIL iRepeats < 0 END_REPEAT;

	F_ByteSwap := USINT_TO_INT(iSize);

ELSE
	(* swap only in the dstData (source unchanged) *)
	pSrcAdrPtr	:= pSrcAdr;
	iTypeSize	:= F_GetPDTypeSize(eType);
	iRepeats	:= 0;
	bEven		:= FALSE;
	bOdd		:= FALSE;

	IF iTypeSize <> 0 THEN
		IF (iSize = iTypeSize) THEN
			(* single element *)
			pDstAdrPtr	:= pDstAdr + USINT_TO_DWORD(iSize - 1);
		ELSIF iSize > iTypeSize THEN
			pDstAdrPtr	:= pDstAdr + USINT_TO_DWORD(iTypeSize - 1);
			iRepeats	:= iSize / iTypeSize - 1;

			IF iRepeats < 0 THEN
				iRepeats := 0;
			END_IF

			IF (iSize MOD iTypeSize) = 0 THEN
				(* array, n-times element size matches block size *)
				bEven := TRUE;
			ELSE
				(* array, n-times element size does not match block size *)
				bOdd := TRUE;
			END_IF
		ELSE
			(* treat as single element *)
			pDstAdrPtr	:= pDstAdr + USINT_TO_DWORD(iSize - 1);
			iTypeSize	:= iSize;
		END_IF
	ELSE
		(* treat as single element *)
		pDstAdrPtr	:= pDstAdr + USINT_TO_DWORD(iSize - 1);
		iTypeSize	:= iSize;
	END_IF

	pSrcAdrPtrOrg	:= pSrcAdrPtr;
	pDstAdrPtrOrg	:= pDstAdrPtr;

	(* execute at least once *)
	REPEAT
		FOR iIndex := 0 TO iTypeSize-1 DO
			pDstAdrPtr^	:= pSrcAdrPtr^;
			pSrcAdrPtr	:= pSrcAdrPtr + DWORD#1;
			pDstAdrPtr	:= pDstAdrPtr - DWORD#1;
		END_FOR

		IF bEven OR bOdd THEN
			pSrcAdrPtr		:= pSrcAdrPtrOrg + USINT_TO_DWORD(iTypeSize);
			pSrcAdrPtrOrg	:= pSrcAdrPtr;
			pDstAdrPtr		:= pDstAdrPtrOrg + USINT_TO_DWORD(iTypeSize);
			pDstAdrPtrOrg	:= pDstAdrPtr;
		END_IF

		iRepeats := iRepeats - 1;
	UNTIL iRepeats < 0 END_REPEAT;

	F_ByteSwap := USINT_TO_INT(iSize);
END_IF
END_FUNCTION

(* POU F_GetPDTypeSize, ST *)
FUNCTION F_GetPDTypeSize : USINT
(*****************************************************************************************************************
	DESCRIPTION:	This FUNCTION returns data size of values in a DPV1 Read Telegram

	CHANGE LOG:
	BY		DATE		DESCRIPTION OF CHANGE
	ICh		2006/08/09	Bugfix for Error
	ICh		2006/07/10	enhanced error reporting
	ICh		2006/07/05	First Version

******************************************************************************************************************)
VAR_INPUT
	eFormat				: E_PD_Datatype;
END_VAR
VAR
END_VAR
CASE eFormat OF
	ePD_BOOL, 			(* 0/1 *)
	ePD_INT08, 			(* -128 .. 127 *)
	ePD_UINT08, 		(* 0 .. 255 *)
	ePD_BYTE 			(* 0 .. 255 *)
	 					: F_GetPDTypeSize := 1;

	ePD_INT16, 			(* -32768 .. 32767 *)
	ePD_UINT16, 		(* 0 .. 65535 *)
	ePD_N2_16BIT,
	ePD_T2_TC_16BIT,
	ePD_E2_FIXPT_16,
	ePD_X2_NV_16,
	ePD_WORD,
	ePD_ERROR 			: F_GetPDTypeSize := 2;

	ePD_INT32, 			(* -2147483648 .. 2147483647 *)
	ePD_UINT32, 		(* 0 .. 4294967295 *)
	ePD_FLOAT, 			(* IEEE 754 *)
	ePD_N4_32BIT,
	ePD_T2_TC_32BIT,
	ePD_C2_FIXPT_32,
	ePD_X4_NV_32,
	ePD_TIMEOFDAY_NODI, (* 0 .. 268435455 ms *)
	ePD_TIMEDIFF_NODI, 	(* 0 .. 4294967295 ms *)
	ePD_DWORD			: F_GetPDTypeSize := 4;

	ePD_TIMEOFDAY_WDI, (* 6 Bytes:
							4 bytes ms 
							+ 2 bytes day since 1.1.1984 *)
	ePD_TIMEDIFF,		(* 4|6 Bytes:
							4 bytes ms 
							+ optional 2 bytes days *)
	ePD_TIMEDIFF_WDI	: F_GetPDTypeSize := 6; (* 6 Bytes:
							4 bytes ms 
							+ 2 bytes days *)

	ePD_DATE			: F_GetPDTypeSize := 7; (* 7 Bytes:
							2 bytes ms
							+ 2 bits (res.), 6 bits (minutes) 
							+ 1 bit (0: StdTime/1: DaylightSavingTime), 2 bits (res.), 5 bits (hours) 
							+ 3 bits (DayOfWeek), 5 bits (DayOfMonth) 
							+ 2 bits (res.), 6 bits (month) 
							+ 1 bit (res.), 7 bits (year) *)

ELSE
(*
	ePD_VSTRING,
	ePD_OCTSTRING,
	ePD_V2_BITSEQ,
	ePD_L2_NIBBLE,
	ePD_R2_RECIP_TC,
	ePD_D2_TC,
	ePD_ZERO,			: F_GetPDTypeSize := 0;
*)

	F_GetPDTypeSize := 0;
END_CASE
END_FUNCTION

(* POU F_CheckForSwapBytes, ST *)
FUNCTION F_CheckForSwapBytes : BOOL
(*****************************************************************************************************************
	DESCRIPTION:	This FUNCTION checks for byte swapping for data in a value of a DPV1 Read Telegram

	CHANGE LOG:
	BY		DATE		DESCRIPTION OF CHANGE
	ICh		2006/08/09	Bugfix for Error
	ICh		2006/07/05	First Version

******************************************************************************************************************)
VAR_INPUT
	eFormat				: E_PD_Datatype;
END_VAR
VAR
END_VAR
CASE eFormat OF
	ePD_INT16, 			(* -32768 .. 32767 *)
	ePD_UINT16, 		(* 0 .. 65535 *)
	ePD_N2_16BIT,
	ePD_T2_TC_16BIT,
	ePD_E2_FIXPT_16,
	ePD_X2_NV_16,
	ePD_WORD,
	ePD_ERROR 			: F_CheckForSwapBytes := TRUE;

	ePD_INT32, 			(* -2147483648 .. 2147483647 *)
	ePD_UINT32, 		(* 0 .. 4294967295 *)
	ePD_FLOAT, 			(* IEEE 754 *)
	ePD_N4_32BIT,
	ePD_T2_TC_32BIT,
	ePD_C2_FIXPT_32,
	ePD_X4_NV_32,
	ePD_TIMEOFDAY_NODI, (* 0 .. 268435455 ms *)
	ePD_TIMEDIFF_NODI, 	(* 0 .. 4294967295 ms *)
	ePD_DWORD			: F_CheckForSwapBytes := TRUE;

	ePD_TIMEOFDAY_WDI, (* 6 Bytes:
							4 bytes ms 
							+ 2 bytes day since 1.1.1984 *)
	ePD_TIMEDIFF,		(* 4|6 Bytes:
							4 bytes ms 
							+ optional 2 bytes days *)
	ePD_TIMEDIFF_WDI	: F_CheckForSwapBytes := TRUE; (* 6 Bytes:
							4 bytes ms 
							+ 2 bytes days *)

	ePD_DATE			: F_CheckForSwapBytes := TRUE; (* 7 Bytes:
							2 bytes ms
							+ 2 bits (res.), 6 bits (minutes) 
							+ 1 bit (0: StdTime/1: DaylightSavingTime), 2 bits (res.), 5 bits (hours) 
							+ 3 bits (DayOfWeek), 5 bits (DayOfMonth) 
							+ 2 bits (res.), 6 bits (month) 
							+ 1 bit (res.), 7 bits (year) *)

ELSE
(*
	ePD_VSTRING,
	ePD_OCTSTRING,
	ePD_V2_BITSEQ,
	ePD_L2_NIBBLE,
	ePD_R2_RECIP_TC,
	ePD_D2_TC,
	ePD_ZERO 			: F_CheckForSwapBytes := FALSE;
*)

	F_CheckForSwapBytes := FALSE;
END_CASE
END_FUNCTION

(* POU F_CreateDpv1ReadReqPkg, ST *)
FUNCTION F_CreateDpv1ReadReqPkg : USINT
(*****************************************************************************************************************
	DESCRIPTION:	This FUNCTION creates a DPV1 Read Telegram

	CHANGE LOG:
	BY		DATE		DESCRIPTION OF CHANGE
	ICh		2006/07/10	enhanced error reporting
	ICh		2006/07/05	First Version

******************************************************************************************************************)
VAR_INPUT
	pDpv1ReqData		: POINTER TO ARRAY [1..iMAX_DPV1_SIZE] OF BYTE; (* DPV1 read request *)
	iNumOfParams		: USINT;		(* 1..39;     else: reserved *)
	iDriveId			: USINT;
END_VAR
VAR_IN_OUT
	stDpv1Parameter		: ARRAY [1..iMAX_DPV1_PARAMS] OF ST_Dpv1ParamAddrEx; (* list of parameters *)
END_VAR
VAR
	stDpv1ReqHeader		: ST_Dpv1Header;
	stDpv1ParameterSwap	: ST_Dpv1ParamAddr; (* parameter address with swapped bytes  *)
	iDpv1ReqIndex		: UDINT;
	iPIndex				: INT;
END_VAR
(* clear data *)
MEMSET(pDpv1ReqData, 0, iMAX_DPV1_SIZE);
iDpv1ReqIndex := 0;

IF iNumOfParams >= 1 AND iNumOfParams <= 39 THEN
	(* preset header data *)
	stDpv1ReqHeader.iRequestRef	:= 0; 			 (* USINT *)
	stDpv1ReqHeader.iRequestID	:= 1; 			 (* SINT  *) (* 1: Read;   2: Write;     0x40..0x7F: manufacturer specific;   else: reserved *)
	stDpv1ReqHeader.iAxis		:= iDriveId;     (* USINT *)
	stDpv1ReqHeader.iNumOfParams:= iNumOfParams; (* USINT *)

	MEMCPY(pDpv1ReqData + iDpv1ReqIndex, ADR(stDpv1ReqHeader), SIZEOF(stDpv1ReqHeader));
	iDpv1ReqIndex := iDpv1ReqIndex + SIZEOF(stDpv1ReqHeader);

	(* preset parameter data *)
	FOR iPIndex := 1 TO iNumOfParams DO
		IF iDpv1ReqIndex + SIZEOF(stDpv1ParameterSwap) <= 240 THEN
			stDpv1ParameterSwap.iAttribute 			:= stDpv1Parameter[iPIndex].iAttribute;
			stDpv1ParameterSwap.iNumOfElements 		:= stDpv1Parameter[iPIndex].iNumOfElements;
			stDpv1ParameterSwap.iParameterNumber 	:= stDpv1Parameter[iPIndex].iParameterNumber;
			stDpv1ParameterSwap.iSubIndex 			:= stDpv1Parameter[iPIndex].iSubIndex;

			(* swap bytes of datatypes bigger than 8bit to MOTOROLA format *)
			F_ByteSwap(ADR(stDpv1ParameterSwap.iParameterNumber), ADR(stDpv1ParameterSwap.iParameterNumber), SIZEOF(stDpv1ParameterSwap.iParameterNumber), ePD_UINT16);
			F_ByteSwap(ADR(stDpv1ParameterSwap.iSubIndex), ADR(stDpv1ParameterSwap.iSubIndex), SIZEOF(stDpv1ParameterSwap.iSubIndex), ePD_UINT16);

			(* add to Dpv1 telegram *)
			MEMCPY(pDpv1ReqData + iDpv1ReqIndex, ADR(stDpv1ParameterSwap), SIZEOF(stDpv1ParameterSwap));
			iDpv1ReqIndex := iDpv1ReqIndex + SIZEOF(stDpv1ParameterSwap);
		ELSE
			MEMSET(pDpv1ReqData, 0, iMAX_DPV1_SIZE); (* telegram too big *)
			iDpv1ReqIndex := iDpv1ReqIndex + SIZEOF(stDpv1ParameterSwap);
			EXIT;
		END_IF
	END_FOR
END_IF

F_CreateDpv1ReadReqPkg := UDINT_TO_USINT(iDpv1ReqIndex);
END_FUNCTION

(* POU F_CreateDpv1ReadReqPkgPNET, ST *)
FUNCTION F_CreateDpv1ReadReqPkgPNET : USINT
(*****************************************************************************************************************
	DESCRIPTION:	This FUNCTION creates a DPV1 Read Telegram for Profinet

	CHANGE LOG:
	BY		DATE		DESCRIPTION OF CHANGE
	ICh		2009/07/27	Fix for stDpv1FrameHeader.stPNIORecord.iLength
	ICh		2009/07/23	First Version

******************************************************************************************************************)
VAR_INPUT
	pDpv1ReqData		: POINTER TO ARRAY [1..iMAX_DPV1_SIZE_PNET_REQ] OF BYTE; (* DPV1 read request *)
	iNumOfParams		: USINT;		(* 1..39;     else: reserved *)
	iDriveId			: USINT;
END_VAR
VAR_IN_OUT
	stDpv1Parameter		: ARRAY [1..iMAX_DPV1_PARAMS] OF ST_Dpv1ParamAddrEx; (* list of parameters *)
END_VAR
VAR
	stDpv1FrameHeader	: ST_PNIOConfigRecord;
	stDpv1ReqHeader		: ST_Dpv1Header;
	stDpv1ParameterSwap	: ST_Dpv1ParamAddr; (* parameter address with swapped bytes  *)
	iDpv1ReqIndex		: UDINT;
	iPIndex				: INT;
END_VAR
(* clear data *)
MEMSET(pDpv1ReqData, 0, iMAX_DPV1_SIZE_PNET_REQ);
iDpv1ReqIndex := 0;

IF iNumOfParams >= 1 AND iNumOfParams <= 39 THEN
	(* preset frame header data *)
	stDpv1FrameHeader.iRW						:= 1;			(* UINT *) (* 0: Response; 1: Request *)
	stDpv1FrameHeader.iNumOfAR					:= 0;			(* UINT *)
	stDpv1FrameHeader.iAPI						:= 16#00003A00;	(* UDINT *)
	stDpv1FrameHeader.iSlot						:= iDriveId;	(* UINT *)
	stDpv1FrameHeader.iSubSlot					:= 1;			(* UINT *)
	stDpv1FrameHeader.stPNIORecord.iIndex		:= 16#B02E;		(* UINT *)
	stDpv1FrameHeader.stPNIORecord.iLength		:= 16#0020;		(* UINT *)
	stDpv1FrameHeader.stPNIORecord.iTransfSeq	:= 0;			(* UINT *)
	stDpv1FrameHeader.stPNIORecord.iAligned		:= 0;			(* UINT *)

	MEMCPY(pDpv1ReqData, ADR(stDpv1FrameHeader), SIZEOF(stDpv1FrameHeader));
	iDpv1ReqIndex := SIZEOF(stDpv1FrameHeader);

	(* preset header data *)
	stDpv1ReqHeader.iRequestRef	:= 0; 			 (* USINT *)
	stDpv1ReqHeader.iRequestID	:= 1; 			 (* SINT  *) (* 1: Read;   2: Write;     0x40..0x7F: manufacturer specific;   else: reserved *)
	stDpv1ReqHeader.iAxis		:= iDriveId;     (* USINT *)
	stDpv1ReqHeader.iNumOfParams:= iNumOfParams; (* USINT *)

	MEMCPY(pDpv1ReqData + iDpv1ReqIndex, ADR(stDpv1ReqHeader), SIZEOF(stDpv1ReqHeader));
	iDpv1ReqIndex := iDpv1ReqIndex + SIZEOF(stDpv1ReqHeader);

	(* preset parameter data *)
	FOR iPIndex := 1 TO iNumOfParams DO
		IF iDpv1ReqIndex + SIZEOF(stDpv1ParameterSwap) <= iMAX_DPV1_SIZE_PNET_REQ THEN
			stDpv1ParameterSwap.iAttribute 			:= stDpv1Parameter[iPIndex].iAttribute;
			stDpv1ParameterSwap.iNumOfElements 		:= stDpv1Parameter[iPIndex].iNumOfElements;
			stDpv1ParameterSwap.iParameterNumber 	:= stDpv1Parameter[iPIndex].iParameterNumber;
			stDpv1ParameterSwap.iSubIndex 			:= stDpv1Parameter[iPIndex].iSubIndex;

			(* swap bytes of datatypes bigger than 8bit to MOTOROLA format *)
			F_ByteSwap(ADR(stDpv1ParameterSwap.iParameterNumber), ADR(stDpv1ParameterSwap.iParameterNumber), SIZEOF(stDpv1ParameterSwap.iParameterNumber), ePD_UINT16);
			F_ByteSwap(ADR(stDpv1ParameterSwap.iSubIndex), ADR(stDpv1ParameterSwap.iSubIndex), SIZEOF(stDpv1ParameterSwap.iSubIndex), ePD_UINT16);

			(* add to Dpv1 telegram *)
			MEMCPY(pDpv1ReqData + iDpv1ReqIndex, ADR(stDpv1ParameterSwap), SIZEOF(stDpv1ParameterSwap));
			iDpv1ReqIndex := iDpv1ReqIndex + SIZEOF(stDpv1ParameterSwap);
		ELSE
			MEMSET(pDpv1ReqData, 0, iMAX_DPV1_SIZE_PNET_REQ); (* telegram too big *)
			iDpv1ReqIndex := iDpv1ReqIndex + SIZEOF(stDpv1ParameterSwap);
			EXIT;
		END_IF
	END_FOR

	IF iDpv1ReqIndex <= iMAX_DPV1_SIZE_PNET_REQ  THEN
		stDpv1FrameHeader.stPNIORecord.iLength := UDINT_TO_UINT(iDpv1ReqIndex - SIZEOF(stDpv1FrameHeader));
		MEMCPY(pDpv1ReqData, ADR(stDpv1FrameHeader), SIZEOF(stDpv1FrameHeader));
	END_IF
END_IF

F_CreateDpv1ReadReqPkgPNET := UDINT_TO_USINT(iDpv1ReqIndex);
END_FUNCTION

(* POU F_CreateDpv1WriteReqPkg, ST *)
FUNCTION F_CreateDpv1WriteReqPkg : USINT
(*****************************************************************************************************************
	DESCRIPTION:	This FUNCTION creates a DPV1 Write Telegram

	CHANGE LOG:
	BY		DATE		DESCRIPTION OF CHANGE
	ICh		2007/01/04	stDpv1ValueHeaderEx as VAR_IN_OUT, extended header, extracting values as string
	ICh		2006/07/10	enhanced error reporting
	ICh		2006/07/07	First Version

******************************************************************************************************************)
VAR_INPUT
	pDpv1ReqData		: POINTER TO ARRAY [1..iMAX_DPV1_SIZE] OF BYTE; (* DPV1 write request *)
	iNumOfParams		: USINT;		(* 1..39;     else: reserved *)
	iDriveId			: USINT;
END_VAR
VAR_IN_OUT
	stDpv1Parameter		: ARRAY [1..iMAX_DPV1_PARAMS] OF ST_Dpv1ParamAddrEx; (* list of parameters *)
	stDpv1ValueHeaderEx	: ARRAY [1..iMAX_DPV1_PARAMS] OF ST_Dpv1ValueHeaderEx;
END_VAR
VAR
	stDpv1ReqHeader		: ST_Dpv1Header;
	stDpv1ParameterSwap	: ST_Dpv1ParamAddr; (* parameter address with swapped bytes  *)
	iDpv1ReqIndex		: UDINT;
	iPIndex				: INT;
	stDpv1ValueHeader	: ST_Dpv1ValueHeader;
	iSize				: UDINT;
	bError				: BOOL;
	bAddFillByte		: BOOL;
END_VAR
(* clear header *)
MEMSET(ADR(stDpv1ValueHeaderEx), 0, SIZEOF(stDpv1ValueHeaderEx));

(* clear data *)
MEMSET(pDpv1ReqData, 0, iMAX_DPV1_SIZE);
iDpv1ReqIndex := 0;
bError := FALSE;

IF iNumOfParams >= 1 AND iNumOfParams <= 39 THEN
	(* preset header data *)
	stDpv1ReqHeader.iRequestRef	:= 0; 			 (* USINT *)
	stDpv1ReqHeader.iRequestID	:= 2; 			 (* SINT  *) (* 1: Read;   2: Write;     0x40..0x7F: manufacturer specific;   else: reserved *)
	stDpv1ReqHeader.iAxis		:= iDriveId;     (* USINT *)
	stDpv1ReqHeader.iNumOfParams:= iNumOfParams; (* USINT *)

	MEMCPY(pDpv1ReqData + iDpv1ReqIndex, ADR(stDpv1ReqHeader), SIZEOF(stDpv1ReqHeader));
	iDpv1ReqIndex := iDpv1ReqIndex + SIZEOF(stDpv1ReqHeader);

	(* preset parameter data *)
	FOR iPIndex := 1 TO iNumOfParams DO
		IF iDpv1ReqIndex + SIZEOF(stDpv1ParameterSwap) <= 240 THEN
			stDpv1ParameterSwap.iAttribute 			:= stDpv1Parameter[iPIndex].iAttribute;
			stDpv1ParameterSwap.iNumOfElements 		:= stDpv1Parameter[iPIndex].iNumOfElements;
			stDpv1ParameterSwap.iParameterNumber 	:= stDpv1Parameter[iPIndex].iParameterNumber;
			stDpv1ParameterSwap.iSubIndex 			:= stDpv1Parameter[iPIndex].iSubIndex;

			(* swap bytes of datatypes bigger than 8bit to MOTOROLA format *)
			F_ByteSwap(ADR(stDpv1ParameterSwap.iParameterNumber), ADR(stDpv1ParameterSwap.iParameterNumber), SIZEOF(stDpv1ParameterSwap.iParameterNumber), ePD_UINT16);
			F_ByteSwap(ADR(stDpv1ParameterSwap.iSubIndex), ADR(stDpv1ParameterSwap.iSubIndex), SIZEOF(stDpv1ParameterSwap.iSubIndex), ePD_UINT16);

			(* add to Dpv1 telegram *)
			MEMCPY(pDpv1ReqData + iDpv1ReqIndex, ADR(stDpv1ParameterSwap), SIZEOF(stDpv1ParameterSwap));
			iDpv1ReqIndex := iDpv1ReqIndex + SIZEOF(stDpv1ParameterSwap);
		ELSE
			MEMSET(pDpv1ReqData, 0, iMAX_DPV1_SIZE); (* telegram too big *)
			iDpv1ReqIndex := iDpv1ReqIndex + SIZEOF(stDpv1ParameterSwap);
			bError	:= TRUE;
			EXIT;
		END_IF
	END_FOR


	(* preset parameter values *)
	IF NOT bError THEN
		FOR iPIndex := 1 TO iNumOfParams DO
			IF ((stDpv1Parameter[iPIndex].iNumOfValues * F_GetPDTypeSize(stDpv1Parameter[iPIndex].eFormat)) MOD 2) = 0 THEN
				iSize := stDpv1Parameter[iPIndex].iNumOfValues * F_GetPDTypeSize(stDpv1Parameter[iPIndex].eFormat);
				bAddFillByte := FALSE;
			ELSE
				iSize := stDpv1Parameter[iPIndex].iNumOfValues * F_GetPDTypeSize(stDpv1Parameter[iPIndex].eFormat) + 1;
				bAddFillByte := TRUE;
			END_IF

			IF iDpv1ReqIndex + SIZEOF(stDpv1ValueHeader) + iSize <= 240 THEN
				stDpv1ValueHeader.iFormat	 				:= INT_TO_USINT(stDpv1Parameter[iPIndex].eFormat);
				stDpv1ValueHeader.iNumOfValues 				:= UINT_TO_USINT(stDpv1Parameter[iPIndex].iNumOfValues);

				stDpv1ValueHeaderEx[iPIndex].eFormat 		:= stDpv1Parameter[iPIndex].eFormat;
				stDpv1ValueHeaderEx[iPIndex].iNumOfValues 	:= stDpv1ValueHeader.iNumOfValues;
				stDpv1ValueHeaderEx[iPIndex].iOffset 		:= UDINT_TO_USINT(iDpv1ReqIndex);
				stDpv1ValueHeaderEx[iPIndex].iDataLen 		:= UDINT_TO_UINT(iSize);
				stDpv1ValueHeaderEx[iPIndex].strData  		:= F_GetDataString(stDpv1ValueHeaderEx[iPIndex].eFormat,
					stDpv1ValueHeaderEx[iPIndex].iNumOfValues, stDpv1Parameter[iPIndex].iDataAddr, iSize);

				(* add header to Dpv1 telegram *)
				MEMCPY(pDpv1ReqData + iDpv1ReqIndex, ADR(stDpv1ValueHeader), SIZEOF(stDpv1ValueHeader));
				iDpv1ReqIndex := iDpv1ReqIndex + SIZEOF(stDpv1ValueHeader);

				(* add value(s) to Dpv1 telegram *)
				MEMCPY(pDpv1ReqData + iDpv1ReqIndex, stDpv1Parameter[iPIndex].iDataAddr, stDpv1Parameter[iPIndex].iDataSize);
				IF F_CheckForSwapBytes(stDpv1Parameter[iPIndex].eFormat) THEN
					(* swap bytes of datatypes bigger than 8bit to MOTOROLA format *)
					F_ByteSwap(pDpv1ReqData + iDpv1ReqIndex, pDpv1ReqData + iDpv1ReqIndex, UDINT_TO_USINT(stDpv1Parameter[iPIndex].iDataSize), stDpv1Parameter[iPIndex].eFormat);
				END_IF
				iDpv1ReqIndex := iDpv1ReqIndex + iSize;

				IF bAddFillByte THEN
					MEMSET(pDpv1ReqData + iDpv1ReqIndex - 1, 0, 1);
					bAddFillByte := FALSE;
				END_IF
			ELSE
				MEMSET(pDpv1ReqData, 0, iMAX_DPV1_SIZE); (* telegram too big *)
				iDpv1ReqIndex := iDpv1ReqIndex + SIZEOF(stDpv1ValueHeader) + iSize;
				EXIT;
			END_IF
		END_FOR
	END_IF
END_IF

F_CreateDpv1WriteReqPkg := UDINT_TO_USINT(iDpv1ReqIndex);
END_FUNCTION

(* POU F_GetDataString, ST *)
FUNCTION F_GetDataString : STRING
VAR_INPUT
	eFormat				: E_PD_Datatype;
	iNumOfValues		: USINT;	(* 0..234: number of values;   else: reserved *)
	iDataAddr			: UDINT;	(* address of buffer/address of plc variable *)
	iDataSize			: UDINT;	(* size of buffer/size of plc variable *)
END_VAR
VAR
	iIdx				: INT;
	iInt32				: DINT;
	iUInt32				: UDINT;
	fFloat32			: REAL;
	strRetVal			: STRING;
	iValueSize			: INT;
	iValueAddr			: UDINT;
END_VAR
strRetVal	:= '';
iValueSize	:= F_GetPDTypeSize(eFormat);

FOR iIdx := 1 TO iNumOfValues DO
	CASE eFormat OF
		ePD_INT08,
		ePD_INT16,
		ePD_INT32:
			iValueAddr := iDataAddr  + ((iIdx - 1) * iValueSize);
			iInt32 := 0;
			IF iValueAddr + MIN(SIZEOF(iInt32), iValueSize) <= iDataAddr + iDataSize THEN
				MEMCPY(
					ADR(iInt32),
					iValueAddr,
					MIN(SIZEOF(iInt32), iValueSize)
				);
			END_IF
			strRetVal := CONCAT(strRetVal, DINT_TO_STRING(iInt32));

		ePD_UINT08,
		ePD_UINT16,
		ePD_N2_16BIT,
		ePD_T2_TC_16BIT,
		ePD_E2_FIXPT_16,
		ePD_X2_NV_16,
		ePD_WORD,
		ePD_DWORD,
		ePD_ERROR,
		ePD_TIMEOFDAY_NODI,
		ePD_TIMEDIFF_NODI,
		ePD_UINT32:
			iValueAddr := iDataAddr  + ((iIdx - 1) * iValueSize);
			iUInt32 := 0;
			IF iValueAddr + MIN(SIZEOF(iUInt32), iValueSize) <= iDataAddr + iDataSize THEN
				MEMCPY(
					ADR(iUInt32),
					iValueAddr,
					MIN(SIZEOF(iUInt32), iValueSize)
				);
			END_IF
			strRetVal := CONCAT(strRetVal, UDINT_TO_STRING(iUInt32));

		ePD_FLOAT: 			(* IEEE 754 *)
			iValueAddr := iDataAddr  + ((iIdx - 1) * iValueSize);
			fFloat32 := 0;
			IF iValueAddr + MIN(SIZEOF(fFloat32), iValueSize) <= iDataAddr + iDataSize THEN
				MEMCPY(
					ADR(fFloat32),
					iValueAddr,
					MIN(SIZEOF(fFloat32), iValueSize)
				);
			END_IF
			strRetVal := CONCAT(strRetVal, REAL_TO_STRING(fFloat32));

	ELSE

		F_GetDataString := 'See Data';
		EXIT;
	END_CASE

	IF iIdx < iNumOfValues THEN
		strRetVal := CONCAT(strRetVal, '; ');
	END_IF
END_FOR

F_GetDataString := strRetVal;
END_FUNCTION

(* POU F_CreateDpv1WriteReqPkgPNET, ST *)
FUNCTION F_CreateDpv1WriteReqPkgPNET : USINT
(*****************************************************************************************************************
	DESCRIPTION:	This FUNCTION creates a DPV1 Write Telegram for Profinet

	CHANGE LOG:
	BY		DATE		DESCRIPTION OF CHANGE
	ICh		2009/07/27	Fix for stDpv1FrameHeader.stPNIORecord.iLength
	ICh		2009/07/23	First Version

******************************************************************************************************************)
VAR_INPUT
	pDpv1ReqData		: POINTER TO ARRAY [1..iMAX_DPV1_SIZE_PNET_REQ] OF BYTE; (* DPV1 write request *)
	iNumOfParams		: USINT;		(* 1..39;     else: reserved *)
	iDriveId			: USINT;
END_VAR
VAR_IN_OUT
	stDpv1Parameter		: ARRAY [1..iMAX_DPV1_PARAMS] OF ST_Dpv1ParamAddrEx; (* list of parameters *)
	stDpv1ValueHeaderEx	: ARRAY [1..iMAX_DPV1_PARAMS] OF ST_Dpv1ValueHeaderEx;
END_VAR
VAR
	stDpv1FrameHeader	: ST_PNIOConfigRecord;
	stDpv1ReqHeader		: ST_Dpv1Header;
	stDpv1ParameterSwap	: ST_Dpv1ParamAddr; (* parameter address with swapped bytes  *)
	iDpv1ReqIndex		: UDINT;
	iPIndex				: INT;
	stDpv1ValueHeader	: ST_Dpv1ValueHeader;
	iSize				: UDINT;
	bError				: BOOL;
	bAddFillByte		: BOOL;
END_VAR
(* clear header *)
MEMSET(ADR(stDpv1ValueHeaderEx), 0, SIZEOF(stDpv1ValueHeaderEx));

(* clear data *)
MEMSET(pDpv1ReqData, 0, iMAX_DPV1_SIZE_PNET_REQ);
iDpv1ReqIndex := 0;
bError := FALSE;

IF iNumOfParams >= 1 AND iNumOfParams <= 39 THEN
	(* preset frame header data *)
	stDpv1FrameHeader.iRW						:= 1;			(* UINT *) (* 0: Response; 1: Request *)
	stDpv1FrameHeader.iNumOfAR					:= 0;			(* UINT *)
	stDpv1FrameHeader.iAPI						:= 16#00003A00;	(* UDINT *)
	stDpv1FrameHeader.iSlot						:= iDriveId;	(* UINT *)
	stDpv1FrameHeader.iSubSlot					:= 1;			(* UINT *)
	stDpv1FrameHeader.stPNIORecord.iIndex		:= 16#B02E;		(* UINT *)
	stDpv1FrameHeader.stPNIORecord.iLength		:= 16#0020;		(* UINT *)
	stDpv1FrameHeader.stPNIORecord.iTransfSeq	:= 0;			(* UINT *)
	stDpv1FrameHeader.stPNIORecord.iAligned		:= 0;			(* UINT *)

	MEMCPY(pDpv1ReqData, ADR(stDpv1FrameHeader), SIZEOF(stDpv1FrameHeader));
	iDpv1ReqIndex := SIZEOF(stDpv1FrameHeader);

	(* preset header data *)
	stDpv1ReqHeader.iRequestRef	:= 0; 			 (* USINT *)
	stDpv1ReqHeader.iRequestID	:= 2; 			 (* SINT  *) (* 1: Read;   2: Write;     0x40..0x7F: manufacturer specific;   else: reserved *)
	stDpv1ReqHeader.iAxis		:= iDriveId;     (* USINT *)
	stDpv1ReqHeader.iNumOfParams:= iNumOfParams; (* USINT *)

	MEMCPY(pDpv1ReqData + iDpv1ReqIndex, ADR(stDpv1ReqHeader), SIZEOF(stDpv1ReqHeader));
	iDpv1ReqIndex := iDpv1ReqIndex + SIZEOF(stDpv1ReqHeader);

	(* preset parameter data *)
	FOR iPIndex := 1 TO iNumOfParams DO
		IF iDpv1ReqIndex + SIZEOF(stDpv1ParameterSwap) <= iMAX_DPV1_SIZE_PNET_REQ THEN
			stDpv1ParameterSwap.iAttribute 			:= stDpv1Parameter[iPIndex].iAttribute;
			stDpv1ParameterSwap.iNumOfElements 		:= stDpv1Parameter[iPIndex].iNumOfElements;
			stDpv1ParameterSwap.iParameterNumber 	:= stDpv1Parameter[iPIndex].iParameterNumber;
			stDpv1ParameterSwap.iSubIndex 			:= stDpv1Parameter[iPIndex].iSubIndex;

			(* swap bytes of datatypes bigger than 8bit to MOTOROLA format *)
			F_ByteSwap(ADR(stDpv1ParameterSwap.iParameterNumber), ADR(stDpv1ParameterSwap.iParameterNumber), SIZEOF(stDpv1ParameterSwap.iParameterNumber), ePD_UINT16);
			F_ByteSwap(ADR(stDpv1ParameterSwap.iSubIndex), ADR(stDpv1ParameterSwap.iSubIndex), SIZEOF(stDpv1ParameterSwap.iSubIndex), ePD_UINT16);

			(* add to Dpv1 telegram *)
			MEMCPY(pDpv1ReqData + iDpv1ReqIndex, ADR(stDpv1ParameterSwap), SIZEOF(stDpv1ParameterSwap));
			iDpv1ReqIndex := iDpv1ReqIndex + SIZEOF(stDpv1ParameterSwap);
		ELSE
			MEMSET(pDpv1ReqData, 0, iMAX_DPV1_SIZE_PNET_REQ); (* telegram too big *)
			iDpv1ReqIndex := iDpv1ReqIndex + SIZEOF(stDpv1ParameterSwap);
			bError	:= TRUE;
			EXIT;
		END_IF
	END_FOR


	(* preset parameter values *)
	IF NOT bError THEN
		FOR iPIndex := 1 TO iNumOfParams DO
			IF ((stDpv1Parameter[iPIndex].iNumOfValues * F_GetPDTypeSize(stDpv1Parameter[iPIndex].eFormat)) MOD 2) = 0 THEN
				iSize := stDpv1Parameter[iPIndex].iNumOfValues * F_GetPDTypeSize(stDpv1Parameter[iPIndex].eFormat);
				bAddFillByte := FALSE;
			ELSE
				iSize := stDpv1Parameter[iPIndex].iNumOfValues * F_GetPDTypeSize(stDpv1Parameter[iPIndex].eFormat) + 1;
				bAddFillByte := TRUE;
			END_IF

			IF iDpv1ReqIndex + SIZEOF(stDpv1ValueHeader) + iSize <= iMAX_DPV1_SIZE_PNET_REQ THEN
				stDpv1ValueHeader.iFormat	 				:= INT_TO_USINT(stDpv1Parameter[iPIndex].eFormat);
				stDpv1ValueHeader.iNumOfValues 				:= UINT_TO_USINT(stDpv1Parameter[iPIndex].iNumOfValues);

				stDpv1ValueHeaderEx[iPIndex].eFormat 		:= stDpv1Parameter[iPIndex].eFormat;
				stDpv1ValueHeaderEx[iPIndex].iNumOfValues 	:= stDpv1ValueHeader.iNumOfValues;
				stDpv1ValueHeaderEx[iPIndex].iOffset 		:= UDINT_TO_USINT(iDpv1ReqIndex);
				stDpv1ValueHeaderEx[iPIndex].iDataLen 		:= UDINT_TO_UINT(iSize);
				stDpv1ValueHeaderEx[iPIndex].strData  		:= F_GetDataString(stDpv1ValueHeaderEx[iPIndex].eFormat,
					stDpv1ValueHeaderEx[iPIndex].iNumOfValues, stDpv1Parameter[iPIndex].iDataAddr, iSize);

				(* add header to Dpv1 telegram *)
				MEMCPY(pDpv1ReqData + iDpv1ReqIndex, ADR(stDpv1ValueHeader), SIZEOF(stDpv1ValueHeader));
				iDpv1ReqIndex := iDpv1ReqIndex + SIZEOF(stDpv1ValueHeader);

				(* add value(s) to Dpv1 telegram *)
				MEMCPY(pDpv1ReqData + iDpv1ReqIndex, stDpv1Parameter[iPIndex].iDataAddr, stDpv1Parameter[iPIndex].iDataSize);
				IF F_CheckForSwapBytes(stDpv1Parameter[iPIndex].eFormat) THEN
					(* swap bytes of datatypes bigger than 8bit to MOTOROLA format *)
					F_ByteSwap(pDpv1ReqData + iDpv1ReqIndex, pDpv1ReqData + iDpv1ReqIndex, UDINT_TO_USINT(stDpv1Parameter[iPIndex].iDataSize), stDpv1Parameter[iPIndex].eFormat);
				END_IF
				iDpv1ReqIndex := iDpv1ReqIndex + iSize;

				IF bAddFillByte THEN
					MEMSET(pDpv1ReqData + iDpv1ReqIndex - 1, 0, 1);
					bAddFillByte := FALSE;
				END_IF
			ELSE
				MEMSET(pDpv1ReqData, 0, iMAX_DPV1_SIZE_PNET_REQ); (* telegram too big *)
				iDpv1ReqIndex := iDpv1ReqIndex + SIZEOF(stDpv1ValueHeader) + iSize;
				EXIT;
			END_IF
		END_FOR

		IF iDpv1ReqIndex <= iMAX_DPV1_SIZE_PNET_REQ  THEN
			stDpv1FrameHeader.stPNIORecord.iLength := UDINT_TO_UINT(iDpv1ReqIndex - SIZEOF(stDpv1FrameHeader));
			MEMCPY(pDpv1ReqData, ADR(stDpv1FrameHeader), SIZEOF(stDpv1FrameHeader));
		END_IF
	END_IF
END_IF

F_CreateDpv1WriteReqPkgPNET := UDINT_TO_USINT(iDpv1ReqIndex);
END_FUNCTION

(* POU F_GetVersionTcIoFunctions, ST *)
FUNCTION F_GetVersionTcIoFunctions : UINT	(*Gets the library version info *)
VAR_INPUT
	nVersionElement		:	INT;
END_VAR
(*
	Possible nVersionElement parameter:
	1	:	major number
	2	:	minor number
	3	:	revision number
*)
VAR
END_VAR
(* Version history:
Date			|	Version	|	created with					|	Author		|	Remark
dd.mm.yyyy
-----------------------------------------------------------------------------------------------------------------------------------------------------------------------------------------------------------------
23.10.2001	|	1.0.0		|	TC 2.8 B707					|	Christoph C.	|	first TC 2.8 release
28.28.2002	|	1.0.1		|	TC 2.8 B722					|	Christoph C.	|	FB_NovRamReadWrite function block added
05.07.2002	|	1.0.2		|	TC 2.8 B735					|	Christoph C.	|	IOF_SER_IDN_Read, IOF_SER_IDN_Write, IOF_SER_DRIVE_Backup function blocks added. TcUtilities.lib must be included
16.09.2002	|	1.0.3		|	TC 2.8 B904					|	Christoph C.	|	AX200x Profibus function blocks added
18.09.2002	|	1.0.4		|	TC 2.8 B904					|	Christoph C.	|	IOF_GetDeviceInfoByName function block added
31.10.2002	|	1.0.5		|	TC 2.8 B739					|	Christoph C.	|	Merged changes in AX200x fb's(GS) in AX200x Profibus folder. FB_AX2000_AXACT, FB_AX2000_JogMode, FB_AX2000_Reference fb's moved to internal folder.
31.10.2002	|	1.0.6		|	TC 2.8 B739					|	Christoph C.	|	ASI function blocks added
06.11.2002	|	1.0.7		|	TC 2.8 B739					|	Christoph C.	|	Library project info added
11.11.2002	|	1.0.8		|	TC 2.8 B740					|	Christoph C.	|	IODEVICETYPES enum type extended (new devices added). 
16.01.2003	|	1.0.9		|	TC 2.9 B925 (saved as 2.8)	|	Christoph C.	|	FB_GetDPRAMInfo function block added.
11.03.2003	|	1.0.10		|	TC 2.9 B929 (saved as 2.8)	|	Christoph C.	|	IOF_SER_DRIVE_Reset  function block added.
06.05.2003	|	1.0.11		|	TC 2.9 B940 (saved as 2.8)	|	Christoph C.	|	FB_GetUPSStatus function block added
12.05.2003	|	1.0.12		|	TC 2.9 B940 (saved as 2.8)	|	Christoph C.	|	nPowerFailCnt and dwChargeFlags UPS status info added.
04.07.2003	|	1.0.13		|	TC 2.9 B945 (saved as 2.8)	|	Christoph C.	|	FB_ReadAdsTecSysData function block added
21.07.2003	|	1.0.14		|	TC 2.9 B945 (saved as 2.8)	|	Christoph C.	|	Merged changes in AX200x fb's(GS) ( digital speed mode added )
24.09.2003	|	1.0.15		|	TC 2.9 B947 (saved as 2.8)	|	Itzko Ch.		|	Bugfix for IOF_SER_IDN_Read (initialization of target buffer)
06.10.2003	|	1.0.16		|	TC 2.9 B947 (saved as 2.8)	|	Itzko Ch.		|	Bugfix for IOF_SER_IDN_Read, IOF_SER_IDN_Write (limiting to cbLen); optimizing IOF_SER_IDN_Read
07.10.2003	|	1.0.17		|	TC 2.9 B947 (saved as 2.8)	|	Itzko Ch.		|	Bugfix for IOF_SER_GetPhase, clear Phase only in case of error, create immediately falling edge on READ of ADSREADEX
04.11.2003	|	1.0.18		|	TC 2.9 B947 (saved as 2.8)	|	Christoph C.	|	Merged changes in ASI function blocks (GS)
04.11.2003	|	1.0.19		|	TC 2.10 B1241 (saved as 2.8)|	Christoph C.	|	IODEVICETYPES enum type extended (new devices added). 
06.11.2006	|	1.0.20		|	TC 2.10 B1302 (saved as 2.8)|	Richard K.		|	Added FB_NovRamReadWriteEx to support NOV-RAM of CX9000
20.11.2006	|	1.0.21		|	TC 2.10 B1307 (saved as 2.8)|	Christoph C.	|	FB_AX2000_AXACT.a_RW_PZD type cast compiler warnings fixed
29.01.2007	|	1.0.22		|	TC 2.10 B1307 (saved as 2.8)|	I.Ch.			|	IOF_SER_DRIVE_BackupEx, ST_SercosParamErrList, ST_SercosParamList added; Profibus DPV1 (Sinamics) added
21.02.2007	|	1.0.23		|	TC 2.10 B1307 (saved as 2.8)|	Christoph C.	|	Added FB_GetUPSStatus() function block support for Windows CE (CP69xx...)
28.03.2007	|	1.0.24		|	TC 2.10 B1310 (saved as 2.8)|	I.Ch.			|	IOF_SER_IDN_Read fix for read length of parameters with variable length
29.03.2007	|	1.0.25		|	TC 2.10 B1310 (saved as 2.8)|	I.Ch.			|	IOF_SER_IDN_Read fix for read length of parameters with variable length
23.08.2007	|	1.0.26		|	TC 2.10 B1310 (saved as 2.8)|	Richard K.		|	Bugfix for FB_NovRamReadWriteEx (offsets were not evaluated corrected for Default_access)
02.04.2008	|	1.0.27		|	TC 2.10 B1325 (saved as 2.8)|	I.Ch.			|	delay resend request after fault for 100ms in FB_Dpv1Read/FB_Dpv1Write
11.07.2008	|	1.0.28		|	TC 2.10 B1328 (saved as 2.8)|	I.Ch.			|	IOF_SER_IDN_Read added mode 1 to read function state
16.07.2008	|	1.0.29		|	TC 2.10 B1328 (saved as 2.8)|	I.Ch.,AnK		|	bugfixing IOF_SER_IDN_Read for mode 1 to read function state
27.04.2009	|	1.0.30		|	TC 2.10 B1335 (saved as 2.8)|	I.Ch.			|	update IODEVICETYPES 
16.08.2010	|	2.0.0		|	TC 2.11 B2015				| Christoph C.		|	Branched version of TcIoFunctions.Lib (for Builds 2.11 only), update IODEVICETYPES, IOF_GetBoxCount invalid data size fix, optiomizations in other IOF_xxx... functions. tTimeout-.Inputs initialized with DEFAULT_ADS_TIMEOUT constant.
28.01.2011	|	2.0.1		|	TC 2.11 B2024				| I.Ch.				|	added Profinet DPV1 communication FBs for Sinamics drives
28.01.2011	|	2.0.2		|	TC 2.11 B2024				| I.Ch.				|	renaming of Profinet DPV1 communication FBs for Sinamics drives
*)	
CASE nVersionElement OF
1:	(* major number *)
	F_GetVersionTcIoFunctions := 2;
2:	(* minor number *)
	F_GetVersionTcIoFunctions := 0;
3:	(* revision number *)
	F_GetVersionTcIoFunctions := 2;
ELSE
	F_GetVersionTcIoFunctions := 16#FFFF;
END_CASE
END_FUNCTION

(* POU F_SplitDpv1ReadResPkg, ST *)
FUNCTION F_SplitDpv1ReadResPkg : USINT
(*****************************************************************************************************************
	DESCRIPTION:	This FUNCTION splits a DPV1 Read response Telegram
					Returns the number of used bytes of the DPV1-Response-telegram
					read values are stored at address of "stDpv1Parameter[iPIndex].iDataAddr"
					possible errors are stored in "stDpv1Parameter[iPIndex].iErrorValue"

	CHANGE LOG:
	BY		DATE		DESCRIPTION OF CHANGE
	ICh		2007/01/04	stDpv1ValueHeaderEx as VAR_IN_OUT, extended header, extracting values as string
	ICh		2006/12/13	cleanup
	ICh		2006/08/09	bugfix for error
	ICh		2006/07/10	enhanced error reporting
	ICh		2006/07/06	First Version

******************************************************************************************************************)
VAR_INPUT
	pDpv1ResData		: POINTER TO ARRAY [1..iMAX_DPV1_SIZE] OF BYTE; (* DPV1 read response *)
END_VAR
VAR_IN_OUT
	stDpv1Parameter		: ARRAY [1..iMAX_DPV1_PARAMS] OF ST_Dpv1ParamAddrEx; (* list of parameters *)
	stDpv1ValueHeaderEx	: ARRAY [1..iMAX_DPV1_PARAMS] OF ST_Dpv1ValueHeaderEx;
END_VAR
VAR
	stDpv1ResHeader		: ST_Dpv1Header;
	stDpv1ValueHeader	: ST_Dpv1ValueHeader;
	iPIndex				: INT;
	iVIndex				: DINT;
	iSize				: USINT;
	eDpv1Error			: E_PD_Dpv1Error;
END_VAR
(* clear header *)
MEMSET(ADR(stDpv1ValueHeaderEx), 0, SIZEOF(stDpv1ValueHeaderEx));

(* get response header *)
MEMCPY(ADR(stDpv1ResHeader), pDpv1ResData, SIZEOF(stDpv1ResHeader));
iVIndex := SIZEOF(stDpv1ResHeader);

FOR iPIndex := 1 TO stDpv1ResHeader.iNumOfParams DO
	(* get value header *)
	MEMCPY(ADR(stDpv1ValueHeader), pDpv1ResData + iVIndex, 2);
	stDpv1ValueHeaderEx[iPIndex].eFormat 		:= USINT_TO_INT(stDpv1ValueHeader.iFormat);
	stDpv1ValueHeaderEx[iPIndex].iNumOfValues 	:= stDpv1ValueHeader.iNumOfValues;
	iVIndex := iVIndex + 2;

	IF stDpv1ValueHeaderEx[iPIndex].iNumOfValues <> 0 THEN
		stDpv1ValueHeaderEx[iPIndex].iOffset := DINT_TO_USINT(iVIndex) + 1;
		stDpv1Parameter[iPIndex].iErrorValue := 0;
		stDpv1Parameter[iPIndex].stError.bError := FALSE;
		stDpv1Parameter[iPIndex].stError.eErrorId := 0;

		IF ((stDpv1ValueHeaderEx[iPIndex].iNumOfValues * F_GetPDTypeSize(stDpv1ValueHeaderEx[iPIndex].eFormat)) MOD 2) = 0 THEN
			iVIndex := iVIndex + stDpv1ValueHeaderEx[iPIndex].iNumOfValues * F_GetPDTypeSize(stDpv1ValueHeaderEx[iPIndex].eFormat);
		ELSE
			iVIndex := iVIndex + stDpv1ValueHeaderEx[iPIndex].iNumOfValues * F_GetPDTypeSize(stDpv1ValueHeaderEx[iPIndex].eFormat) + 1;
		END_IF

		IF stDpv1ValueHeaderEx[iPIndex].eFormat <> ePD_ERROR THEN
			(* OK *)
			iSize := MIN(UDINT_TO_SINT(stDpv1Parameter[iPIndex].iDataSize),
					(F_GetPDTypeSize(stDpv1ValueHeaderEx[iPIndex].eFormat) * stDpv1ValueHeaderEx[iPIndex].iNumOfValues));
			stDpv1ValueHeaderEx[iPIndex].iDataLen := iSize;

			(* get value(s) *)
			MEMCPY(
				stDpv1Parameter[iPIndex].iDataAddr,
				pDpv1ResData + USINT_TO_UDINT(stDpv1ValueHeaderEx[iPIndex].iOffset) - 1,
				iSize
			);

			IF F_CheckForSwapBytes(stDpv1ValueHeaderEx[iPIndex].eFormat) THEN
				(* swap bytes of datatypes bigger than 8bit to INTEL format *)
				F_ByteSwap(stDpv1Parameter[iPIndex].iDataAddr, stDpv1Parameter[iPIndex].iDataAddr, iSize, stDpv1ValueHeaderEx[iPIndex].eFormat);
			END_IF

			stDpv1ValueHeaderEx[iPIndex].strData := F_GetDataString(stDpv1ValueHeaderEx[iPIndex].eFormat,
				stDpv1ValueHeaderEx[iPIndex].iNumOfValues, stDpv1Parameter[iPIndex].iDataAddr, iSize);
		ELSE
			(* error response *)
			iSize := MIN(UDINT_TO_SINT(SIZEOF(stDpv1Parameter[iPIndex].iErrorValue)),
					(F_GetPDTypeSize(stDpv1ValueHeaderEx[iPIndex].eFormat) * stDpv1ValueHeaderEx[iPIndex].iNumOfValues));
			stDpv1ValueHeaderEx[iPIndex].iDataLen := iSize;

			(* get error value *)
			MEMCPY(
				ADR(stDpv1Parameter[iPIndex].iErrorValue),
				pDpv1ResData + USINT_TO_UDINT(stDpv1ValueHeaderEx[iPIndex].iOffset) - 1,
				iSize
			);

			IF F_CheckForSwapBytes(stDpv1ValueHeaderEx[iPIndex].eFormat) THEN
				(* swap bytes of datatypes bigger than 8bit to INTEL format *)
				F_ByteSwap(ADR(stDpv1Parameter[iPIndex].iErrorValue), ADR(stDpv1Parameter[iPIndex].iErrorValue), iSize, stDpv1ValueHeaderEx[iPIndex].eFormat);
			END_IF

			stDpv1Parameter[iPIndex].stError.bError := TRUE;
			stDpv1Parameter[iPIndex].stError.eErrorId := UDINT_TO_INT(stDpv1Parameter[iPIndex].iErrorValue);
			eDpv1Error := stDpv1Parameter[iPIndex].stError.eErrorId;
			stDpv1ValueHeaderEx[iPIndex].strData := INT_TO_STRING(eDpv1Error);
			IF stDpv1ValueHeaderEx[iPIndex].iNumOfValues = 2 THEN
				stDpv1ValueHeaderEx[iPIndex].strData := CONCAT(stDpv1ValueHeaderEx[iPIndex].strData, '; ');
				stDpv1ValueHeaderEx[iPIndex].strData := CONCAT(stDpv1ValueHeaderEx[iPIndex].strData,
						UINT_TO_STRING(UDINT_TO_UINT(SHR(stDpv1Parameter[iPIndex].iErrorValue, 16))));
			END_IF
		END_IF
	ELSE
		stDpv1ValueHeaderEx[iPIndex].iOffset := 0;
		stDpv1ValueHeaderEx[iPIndex].strData := '';
	END_IF

	IF iVIndex >= DINT#239 THEN
		EXIT;
	END_IF
END_FOR

F_SplitDpv1ReadResPkg := DINT_TO_USINT(iVIndex);
END_FUNCTION

(* POU F_SplitDpv1ReadResPkgPNET, ST *)
FUNCTION F_SplitDpv1ReadResPkgPNET : USINT
(*****************************************************************************************************************
	DESCRIPTION:	This FUNCTION splits a DPV1 Read response Telegram for Profinet
					Returns the number of used bytes of the DPV1-Response-telegram
					read values are stored at address of "stDpv1Parameter[iPIndex].iDataAddr"
					possible errors are stored in "stDpv1Parameter[iPIndex].iErrorValue"

	CHANGE LOG:
	BY		DATE		DESCRIPTION OF CHANGE
	ICh		2009/07/23	First Version

******************************************************************************************************************)
VAR_INPUT
	pDpv1ResData		: POINTER TO ARRAY [1..iMAX_DPV1_SIZE_PNET_RES] OF BYTE; (* DPV1 read response *)
END_VAR
VAR_IN_OUT
	stDpv1Parameter		: ARRAY [1..iMAX_DPV1_PARAMS] OF ST_Dpv1ParamAddrEx; (* list of parameters *)
	stDpv1ValueHeaderEx	: ARRAY [1..iMAX_DPV1_PARAMS] OF ST_Dpv1ValueHeaderEx;
END_VAR
VAR
	stDpv1ResHeader		: ST_Dpv1Header;
	stDpv1ValueHeader	: ST_Dpv1ValueHeader;
	iPIndex				: INT;
	iVIndex				: DINT;
	iSize				: USINT;
	eDpv1Error			: E_PD_Dpv1Error;
END_VAR
(* clear header *)
MEMSET(ADR(stDpv1ValueHeaderEx), 0, SIZEOF(stDpv1ValueHeaderEx));

(* get response header *)
MEMCPY(ADR(stDpv1ResHeader), pDpv1ResData, SIZEOF(stDpv1ResHeader));
iVIndex := SIZEOF(stDpv1ResHeader);

FOR iPIndex := 1 TO stDpv1ResHeader.iNumOfParams DO
	(* get value header *)
	MEMCPY(ADR(stDpv1ValueHeader), pDpv1ResData + iVIndex, 2);
	stDpv1ValueHeaderEx[iPIndex].eFormat 		:= USINT_TO_INT(stDpv1ValueHeader.iFormat);
	stDpv1ValueHeaderEx[iPIndex].iNumOfValues 	:= stDpv1ValueHeader.iNumOfValues;
	iVIndex := iVIndex + 2;

	IF stDpv1ValueHeaderEx[iPIndex].iNumOfValues <> 0 THEN
		stDpv1ValueHeaderEx[iPIndex].iOffset := DINT_TO_USINT(iVIndex) + 1;
		stDpv1Parameter[iPIndex].iErrorValue := 0;
		stDpv1Parameter[iPIndex].stError.bError := FALSE;
		stDpv1Parameter[iPIndex].stError.eErrorId := 0;

		IF ((stDpv1ValueHeaderEx[iPIndex].iNumOfValues * F_GetPDTypeSize(stDpv1ValueHeaderEx[iPIndex].eFormat)) MOD 2) = 0 THEN
			iVIndex := iVIndex + stDpv1ValueHeaderEx[iPIndex].iNumOfValues * F_GetPDTypeSize(stDpv1ValueHeaderEx[iPIndex].eFormat);
		ELSE
			iVIndex := iVIndex + stDpv1ValueHeaderEx[iPIndex].iNumOfValues * F_GetPDTypeSize(stDpv1ValueHeaderEx[iPIndex].eFormat) + 1;
		END_IF

		IF stDpv1ValueHeaderEx[iPIndex].eFormat <> ePD_ERROR THEN
			(* OK *)
			iSize := MIN(UDINT_TO_SINT(stDpv1Parameter[iPIndex].iDataSize),
					(F_GetPDTypeSize(stDpv1ValueHeaderEx[iPIndex].eFormat) * stDpv1ValueHeaderEx[iPIndex].iNumOfValues));
			stDpv1ValueHeaderEx[iPIndex].iDataLen := iSize;

			(* get value(s) *)
			MEMCPY(
				stDpv1Parameter[iPIndex].iDataAddr,
				pDpv1ResData + USINT_TO_UDINT(stDpv1ValueHeaderEx[iPIndex].iOffset) - 1,
				iSize
			);

			IF F_CheckForSwapBytes(stDpv1ValueHeaderEx[iPIndex].eFormat) THEN
				(* swap bytes of datatypes bigger than 8bit to INTEL format *)
				F_ByteSwap(stDpv1Parameter[iPIndex].iDataAddr, stDpv1Parameter[iPIndex].iDataAddr, iSize, stDpv1ValueHeaderEx[iPIndex].eFormat);
			END_IF

			stDpv1ValueHeaderEx[iPIndex].strData := F_GetDataString(stDpv1ValueHeaderEx[iPIndex].eFormat,
				stDpv1ValueHeaderEx[iPIndex].iNumOfValues, stDpv1Parameter[iPIndex].iDataAddr, iSize);
		ELSE
			(* error response *)
			iSize := MIN(UDINT_TO_SINT(SIZEOF(stDpv1Parameter[iPIndex].iErrorValue)),
					(F_GetPDTypeSize(stDpv1ValueHeaderEx[iPIndex].eFormat) * stDpv1ValueHeaderEx[iPIndex].iNumOfValues));
			stDpv1ValueHeaderEx[iPIndex].iDataLen := iSize;

			(* get error value *)
			MEMCPY(
				ADR(stDpv1Parameter[iPIndex].iErrorValue),
				pDpv1ResData + USINT_TO_UDINT(stDpv1ValueHeaderEx[iPIndex].iOffset) - 1,
				iSize
			);

			IF F_CheckForSwapBytes(stDpv1ValueHeaderEx[iPIndex].eFormat) THEN
				(* swap bytes of datatypes bigger than 8bit to INTEL format *)
				F_ByteSwap(ADR(stDpv1Parameter[iPIndex].iErrorValue), ADR(stDpv1Parameter[iPIndex].iErrorValue), iSize, stDpv1ValueHeaderEx[iPIndex].eFormat);
			END_IF

			stDpv1Parameter[iPIndex].stError.bError := TRUE;
			stDpv1Parameter[iPIndex].stError.eErrorId := UDINT_TO_INT(stDpv1Parameter[iPIndex].iErrorValue);
			eDpv1Error := stDpv1Parameter[iPIndex].stError.eErrorId;
			stDpv1ValueHeaderEx[iPIndex].strData := INT_TO_STRING(eDpv1Error);
			IF stDpv1ValueHeaderEx[iPIndex].iNumOfValues = 2 THEN
				stDpv1ValueHeaderEx[iPIndex].strData := CONCAT(stDpv1ValueHeaderEx[iPIndex].strData, '; ');
				stDpv1ValueHeaderEx[iPIndex].strData := CONCAT(stDpv1ValueHeaderEx[iPIndex].strData,
						UINT_TO_STRING(UDINT_TO_UINT(SHR(stDpv1Parameter[iPIndex].iErrorValue, 16))));
			END_IF
		END_IF
	ELSE
		stDpv1ValueHeaderEx[iPIndex].iOffset := 0;
		stDpv1ValueHeaderEx[iPIndex].strData := '';
	END_IF

	IF iVIndex >= iMAX_DPV1_SIZE_PNET_RES-1 THEN
		EXIT;
	END_IF
END_FOR

F_SplitDpv1ReadResPkgPNET := DINT_TO_USINT(iVIndex);
END_FUNCTION

(* POU F_SplitDpv1WriteResPkg, ST *)
FUNCTION F_SplitDpv1WriteResPkg : USINT
(*****************************************************************************************************************
	DESCRIPTION:	This FUNCTION splits a DPV1 write response Telegram
					Returns the number of used bytes of the DPV1-Response-telegram
					possible errors are stored in "stDpv1Parameter[iPIndex].iErrorValue"


	CHANGE LOG:
	BY		DATE		DESCRIPTION OF CHANGE
	ICh		2007/01/04	stDpv1ValueHeaderEx as VAR_IN_OUT, extracting values as string
	ICh		2006/12/13	cleanup
	ICh		2006/08/09	bugfix for error
	ICh		2006/07/10	enhanced error reporting
	ICh		2006/07/07	First Version

******************************************************************************************************************)
VAR_INPUT
	pDpv1ResData		: POINTER TO ARRAY [1..iMAX_DPV1_SIZE] OF BYTE; (* DPV1 write response *)
END_VAR
VAR_IN_OUT
	stDpv1Parameter		: ARRAY [1..iMAX_DPV1_PARAMS] OF ST_Dpv1ParamAddrEx; (* list of parameters *)
	stDpv1ValueHeaderEx	: ARRAY [1..iMAX_DPV1_PARAMS] OF ST_Dpv1ValueHeaderEx;
END_VAR
VAR
	stDpv1ResHeader		: ST_Dpv1Header;
	stDpv1ValueHeader	: ST_Dpv1ValueHeader;
	iPIndex				: INT;
	iVIndex				: DINT;
	iSize				: USINT;
	eDpv1Error			: E_PD_Dpv1Error;
	stDpv1ValueHeaderExInt	: ARRAY [1..iMAX_DPV1_PARAMS] OF ST_Dpv1ValueHeaderEx;
END_VAR
(* clear header *)
MEMSET(ADR(stDpv1ValueHeaderExInt), 0, SIZEOF(stDpv1ValueHeaderExInt));

(* get response header *)
MEMCPY(ADR(stDpv1ResHeader), pDpv1ResData, SIZEOF(stDpv1ResHeader));
iVIndex := SIZEOF(stDpv1ResHeader);

FOR iPIndex := 1 TO stDpv1ResHeader.iNumOfParams DO
	(* get value header *)
	MEMCPY(ADR(stDpv1ValueHeader), pDpv1ResData + iVIndex, 2);
	stDpv1ValueHeaderExInt[iPIndex].eFormat 		:= USINT_TO_INT(stDpv1ValueHeader.iFormat);
	stDpv1ValueHeaderExInt[iPIndex].iNumOfValues 	:= stDpv1ValueHeader.iNumOfValues;
	iVIndex := iVIndex + 2;

	IF stDpv1ValueHeaderExInt[iPIndex].iNumOfValues <> 0 THEN
		stDpv1ValueHeaderExInt[iPIndex].iOffset := DINT_TO_USINT(iVIndex) + 1;
		stDpv1Parameter[iPIndex].iErrorValue := 0;
		stDpv1Parameter[iPIndex].stError.bError := FALSE;
		stDpv1Parameter[iPIndex].stError.eErrorId := 0;

		IF ((stDpv1ValueHeaderExInt[iPIndex].iNumOfValues * F_GetPDTypeSize(stDpv1ValueHeaderExInt[iPIndex].eFormat)) MOD 2) = 0 THEN
			iVIndex := iVIndex + stDpv1ValueHeaderExInt[iPIndex].iNumOfValues * F_GetPDTypeSize(stDpv1ValueHeaderExInt[iPIndex].eFormat);
		ELSE
			iVIndex := iVIndex + stDpv1ValueHeaderExInt[iPIndex].iNumOfValues * F_GetPDTypeSize(stDpv1ValueHeaderExInt[iPIndex].eFormat) + 1;
		END_IF

		IF stDpv1ValueHeaderExInt[iPIndex].eFormat <> ePD_ERROR THEN
			(* OK - nothing to do *)
			stDpv1ValueHeaderExInt[iPIndex].strData := '';
		ELSE
			(* error response *)
			iSize := MIN(UDINT_TO_SINT(SIZEOF(stDpv1Parameter[iPIndex].iErrorValue)),
					(F_GetPDTypeSize(stDpv1ValueHeaderExInt[iPIndex].eFormat) * stDpv1ValueHeaderExInt[iPIndex].iNumOfValues));
			stDpv1ValueHeaderExInt[iPIndex].iDataLen := iSize;

			(* get error value *)
			MEMCPY(
				ADR(stDpv1Parameter[iPIndex].iErrorValue),
				pDpv1ResData + USINT_TO_UDINT(stDpv1ValueHeaderExInt[iPIndex].iOffset) - 1,
				iSize
			);

			IF F_CheckForSwapBytes(stDpv1ValueHeaderExInt[iPIndex].eFormat) THEN
				(* swap bytes of datatypes bigger than 8bit to INTEL format *)
				F_ByteSwap(ADR(stDpv1Parameter[iPIndex].iErrorValue), ADR(stDpv1Parameter[iPIndex].iErrorValue), iSize, stDpv1ValueHeaderExInt[iPIndex].eFormat);
			END_IF

			stDpv1Parameter[iPIndex].stError.bError := TRUE;
			stDpv1Parameter[iPIndex].stError.eErrorId := UDINT_TO_INT(stDpv1Parameter[iPIndex].iErrorValue);
			eDpv1Error := stDpv1Parameter[iPIndex].stError.eErrorId;
			stDpv1ValueHeaderExInt[iPIndex].strData := INT_TO_STRING(eDpv1Error);

			IF stDpv1ValueHeaderExInt[iPIndex].iNumOfValues = 2 THEN
				stDpv1ValueHeaderExInt[iPIndex].strData := CONCAT(stDpv1ValueHeaderExInt[iPIndex].strData, '; ');
				stDpv1ValueHeaderExInt[iPIndex].strData := CONCAT(stDpv1ValueHeaderExInt[iPIndex].strData,
						UINT_TO_STRING(UDINT_TO_UINT(SHR(stDpv1Parameter[iPIndex].iErrorValue, 16))));
			END_IF

			stDpv1ValueHeaderEx[iPIndex] := stDpv1ValueHeaderExInt[iPIndex];
		END_IF
	ELSE
		stDpv1ValueHeaderExInt[iPIndex].iOffset := 0;
		stDpv1ValueHeaderExInt[iPIndex].strData := '';
	END_IF

	IF iVIndex >= DINT#239 THEN
		EXIT;
	END_IF
END_FOR

F_SplitDpv1WriteResPkg := DINT_TO_USINT(iVIndex);
END_FUNCTION

(* POU F_SplitDpv1WriteResPkgPNET, ST *)
FUNCTION F_SplitDpv1WriteResPkgPNET : USINT
(*****************************************************************************************************************
	DESCRIPTION:	This FUNCTION splits a DPV1 write response Telegram for Profinet
					Returns the number of used bytes of the DPV1-Response-telegram
					possible errors are stored in "stDpv1Parameter[iPIndex].iErrorValue"


	CHANGE LOG:
	BY		DATE		DESCRIPTION OF CHANGE
	ICh		2009/07/23	First Version

******************************************************************************************************************)
VAR_INPUT
	pDpv1ResData		: POINTER TO ARRAY [1..iMAX_DPV1_SIZE_PNET_RES] OF BYTE; (* DPV1 write response *)
END_VAR
VAR_IN_OUT
	stDpv1Parameter		: ARRAY [1..iMAX_DPV1_PARAMS] OF ST_Dpv1ParamAddrEx; (* list of parameters *)
	stDpv1ValueHeaderEx	: ARRAY [1..iMAX_DPV1_PARAMS] OF ST_Dpv1ValueHeaderEx;
END_VAR
VAR
	stDpv1ResHeader		: ST_Dpv1Header;
	stDpv1ValueHeader	: ST_Dpv1ValueHeader;
	iPIndex				: INT;
	iVIndex				: DINT;
	iSize				: USINT;
	eDpv1Error			: E_PD_Dpv1Error;
	stDpv1ValueHeaderExInt	: ARRAY [1..iMAX_DPV1_PARAMS] OF ST_Dpv1ValueHeaderEx;
END_VAR
(* clear header *)
MEMSET(ADR(stDpv1ValueHeaderExInt), 0, SIZEOF(stDpv1ValueHeaderExInt));

(* get response header *)
MEMCPY(ADR(stDpv1ResHeader), pDpv1ResData, SIZEOF(stDpv1ResHeader));
iVIndex := SIZEOF(stDpv1ResHeader);

FOR iPIndex := 1 TO stDpv1ResHeader.iNumOfParams DO
	(* get value header *)
	MEMCPY(ADR(stDpv1ValueHeader), pDpv1ResData + iVIndex, 2);
	stDpv1ValueHeaderExInt[iPIndex].eFormat 		:= USINT_TO_INT(stDpv1ValueHeader.iFormat);
	stDpv1ValueHeaderExInt[iPIndex].iNumOfValues 	:= stDpv1ValueHeader.iNumOfValues;
	iVIndex := iVIndex + 2;

	IF stDpv1ValueHeaderExInt[iPIndex].iNumOfValues <> 0 THEN
		stDpv1ValueHeaderExInt[iPIndex].iOffset := DINT_TO_USINT(iVIndex) + 1;
		stDpv1Parameter[iPIndex].iErrorValue := 0;
		stDpv1Parameter[iPIndex].stError.bError := FALSE;
		stDpv1Parameter[iPIndex].stError.eErrorId := 0;

		IF ((stDpv1ValueHeaderExInt[iPIndex].iNumOfValues * F_GetPDTypeSize(stDpv1ValueHeaderExInt[iPIndex].eFormat)) MOD 2) = 0 THEN
			iVIndex := iVIndex + stDpv1ValueHeaderExInt[iPIndex].iNumOfValues * F_GetPDTypeSize(stDpv1ValueHeaderExInt[iPIndex].eFormat);
		ELSE
			iVIndex := iVIndex + stDpv1ValueHeaderExInt[iPIndex].iNumOfValues * F_GetPDTypeSize(stDpv1ValueHeaderExInt[iPIndex].eFormat) + 1;
		END_IF

		IF stDpv1ValueHeaderExInt[iPIndex].eFormat <> ePD_ERROR THEN
			(* OK - nothing to do *)
			stDpv1ValueHeaderExInt[iPIndex].strData := '';
		ELSE
			(* error response *)
			iSize := MIN(UDINT_TO_SINT(SIZEOF(stDpv1Parameter[iPIndex].iErrorValue)),
					(F_GetPDTypeSize(stDpv1ValueHeaderExInt[iPIndex].eFormat) * stDpv1ValueHeaderExInt[iPIndex].iNumOfValues));
			stDpv1ValueHeaderExInt[iPIndex].iDataLen := iSize;

			(* get error value *)
			MEMCPY(
				ADR(stDpv1Parameter[iPIndex].iErrorValue),
				pDpv1ResData + USINT_TO_UDINT(stDpv1ValueHeaderExInt[iPIndex].iOffset) - 1,
				iSize
			);

			IF F_CheckForSwapBytes(stDpv1ValueHeaderExInt[iPIndex].eFormat) THEN
				(* swap bytes of datatypes bigger than 8bit to INTEL format *)
				F_ByteSwap(ADR(stDpv1Parameter[iPIndex].iErrorValue), ADR(stDpv1Parameter[iPIndex].iErrorValue), iSize, stDpv1ValueHeaderExInt[iPIndex].eFormat);
			END_IF

			stDpv1Parameter[iPIndex].stError.bError := TRUE;
			stDpv1Parameter[iPIndex].stError.eErrorId := UDINT_TO_INT(stDpv1Parameter[iPIndex].iErrorValue);
			eDpv1Error := stDpv1Parameter[iPIndex].stError.eErrorId;
			stDpv1ValueHeaderExInt[iPIndex].strData := INT_TO_STRING(eDpv1Error);

			IF stDpv1ValueHeaderExInt[iPIndex].iNumOfValues = 2 THEN
				stDpv1ValueHeaderExInt[iPIndex].strData := CONCAT(stDpv1ValueHeaderExInt[iPIndex].strData, '; ');
				stDpv1ValueHeaderExInt[iPIndex].strData := CONCAT(stDpv1ValueHeaderExInt[iPIndex].strData,
						UINT_TO_STRING(UDINT_TO_UINT(SHR(stDpv1Parameter[iPIndex].iErrorValue, 16))));
			END_IF

			stDpv1ValueHeaderEx[iPIndex] := stDpv1ValueHeaderExInt[iPIndex];
		END_IF
	ELSE
		stDpv1ValueHeaderExInt[iPIndex].iOffset := 0;
		stDpv1ValueHeaderExInt[iPIndex].strData := '';
	END_IF

	IF iVIndex >= iMAX_DPV1_SIZE_PNET_RES-1 THEN
		EXIT;
	END_IF
END_FOR

F_SplitDpv1WriteResPkgPNET := DINT_TO_USINT(iVIndex);
END_FUNCTION

(* POU FB_ASI_Addressing, ST *)
(*********************************************************************************************************

NAME..............	:	FB_Addressing
DATE...............	:	21.03.2002
AUTHOR........	:	G.Sieder (Beckhoff Industrieelektronik)

DESCRIPTION:	FB to set or change addresses of ASI-slaves 

HISTORY:	
21.03.2002	gs	start coding
03.09.2002	gs	Autoaddressing removed
18.08.2003	gs	new Errorhandling added
*********************************************************************************************************)
FUNCTION_BLOCK FB_ASI_Addressing
VAR_INPUT
	iOldAddress		:BYTE;
	iNewAddress		:BYTE;
	bStart			:BOOL;

END_VAR
VAR_OUTPUT
	bBusy				:BOOL;
	bErr					:BOOL;
	iErrornumber			:DWORD;

END_VAR
VAR_IN_OUT
	stParameterBuffer		:ST_ParameterBuffer;
END_VAR
VAR
	iaddressState	:INT;
	iParametervalue	:DWORD;
	TrigStart			:R_TRIG;
	fbParameterinterface	:FB_ASI_Parameterinterface;

END_VAR
	CASE iaddressState OF

	(*Idle*)
	0:	TrigStart(clk:=bStart);
		IF TrigStart.Q THEN
			bBusy				:=TRUE;
			bErr					:=FALSE;
			iErrornumber			:=0;
			iaddressState		:=1;
		END_IF

	(*Paramatervalue*)
	1:	iParametervalue	:=0;
		iParametervalue	:=SHL((iParametervalue+iNewAddress),8);
		iParametervalue	:=SHL((iParametervalue+iOldAddress),16);
		iParametervalue	:=iParametervalue+16#0701;
		iaddressState	:=2;

	(*wite Parameters to ASI-Master*)
	2:	fbParameterinterface(iParameternumber	:=16#100,
							iParametervalue	:=iParametervalue,
							stParameterBuffer	:=stParameterBuffer,
							bParametermode	:=TRUE,
							bCycleMode		:=FALSE,
							bCommMode		:=FALSE,
							bRegComm		:=FALSE,
							bStart			:=TRUE);
		IF (NOT fbParameterinterface.bBusy)  THEN
			IF fbParameterinterface.bErr THEN
				bErr			:=TRUE;
				iErrornumber	:=fbParameterinterface.iErrornumber;
			ELSIF (fbParameterinterface.iParameterReadvalue AND 16#8000) <>0 THEN
				bErr			:=TRUE;
				iErrornumber	:=SHR((fbParameterinterface.iParameterReadvalue AND 16#FF000000),24);
			END_IF
			fbParameterinterface(bStart			:=FALSE,
							stParameterBuffer	:=stParameterBuffer,);
			iaddressState	:=10;
		END_IF

	(*Quit*)
	10:	bBusy			:=FALSE;
		bStart			:=FALSE;
		iaddressState	:=0;

	ELSE
		;
	END_CASE
END_FUNCTION_BLOCK

(* POU FB_ASI_Parameterinterface, ST *)
(*********************************************************************************************************

NAME..............	:	FB_Parameterinterface
DATE...............	:	21.03.2002
AUTHOR........	:	G.Sieder (Beckhoff Industrieelektronik)

DESCRIPTION:	basic-FB for Read/Write Parameters from/to  ASI-master 

HISTORY:	
21.03.2002	gs	start coding
21.04.2002	gs	adding data-writing (case 1) to a vitual Buffer to realize a multi-instance mode
*********************************************************************************************************)
FUNCTION_BLOCK FB_ASI_Parameterinterface
VAR_INPUT
	iParameternumber		:WORD;
	iParametervalue		:DWORD;
	bHiWord				:BOOL;		(*0:LoWord, 1:HiWord*)
	bmaskAccess		:BOOL;		(*0:usual access, 1:mask access*)
	iParametermask		:WORD;		(*Parametermask if bmaskAccess:=true*)
	bParametermode		:BOOL;		(*0: Read, 1: Write *)
	bCycleMode			:BOOL;		(*0: Acyclic , 1:Cyclic (permanent Read/Write) *)
	bCommMode			:BOOL;		(*0: Parameteraccess, 1: ADS*)
	bRegComm			:BOOL;		(*Registercommunication: 0: Parameteraccess, 1: Registercommunication *)
	bStart				:BOOL;
END_VAR
VAR_OUTPUT
	bBusy				:BOOL;
	bErr					:BOOL;
	iErrornumber			:DWORD;
	iParameterReadvalue	:DWORD;

END_VAR
VAR_IN_OUT
	stParameterBuffer		:ST_ParameterBuffer;
END_VAR
VAR
	iParameterStep		:INT;
	iParameterstate_intern	:WORD;
	iBufferNumber		:INT;
	TimerBuffer			:TON;

END_VAR
CASE iParameterStep OF

		(*Idle*)
	0:	IF bStart THEN
			bBusy				:=TRUE;
			bErr					:=FALSE;
			iErrornumber			:=0;
			iParameterStep		:=1;
		ELSE
			bBusy				:=FALSE;
		END_IF

		(*Write Parameter *)
	1:	iParameterstate_intern	:=0;
		iParameterstate_intern	:=(iParameternumber AND 2#0000000000111111)+(ROL((iParameternumber AND 2#0000001111000000),2));
		iParameterstate_intern	:=iParameterstate_intern+16#4000;
		IF bParametermode THEN
			iParameterstate_intern	:=iParameterstate_intern+16#40;
		END_IF
		IF bCommMode THEN
			iParameterstate_intern	:=iParameterstate_intern+16#8000;
		END_IF
		IF bRegComm THEN
			iParameterstate_intern	:=iParameterstate_intern+16#80;
		END_IF
		IF bHiWord THEN
			iParameterstate_intern	:=iParameterstate_intern+16#1000;
		END_IF
		IF bmaskAccess THEN
			iParameterstate_intern	:=iParameterstate_intern+16#2000;
		END_IF
		(*set Buffercounter*)
		IF stParameterBuffer.icounterState >49 THEN
			stParameterBuffer.icounterState	:=0;
		ELSE
			stParameterBuffer.icounterState	:=stParameterBuffer.icounterState +1;
		END_IF
		(*register the Buffer location*)
		iBufferNumber	:=stParameterBuffer.icounterState;
		(*writing parameterstate to the first free location of ParameterBuffer*)
		stParameterBuffer.ParameterControl[iBufferNumber]	:=iParameterstate_intern;

		IF bmaskAccess THEN
			IF bHiWord THEN
				stParameterBuffer.iParametervalue[iBufferNumber]	:=ROL(((iParametervalue AND 16#FFFF0000)+iParametermask),16);
			ELSE
				stParameterBuffer.iParametervalue[iBufferNumber]	:=ROL(((SHL(iParametervalue,16))+iParametermask),16);
			END_IF
		ELSE
			stParameterBuffer.iParametervalue[iBufferNumber]	:=iParametervalue;
		END_IF
		iParameterStep		:=2;

		(*Read Parameter*)
	2:	TimerBuffer(in:=TRUE,pt:=t#1s);
		IF stParameterBuffer.iParameterStatus[iBufferNumber] <> 0  THEN
			TimerBuffer(in:=FALSE);
			IF ((stParameterBuffer.iParameterStatus[iBufferNumber] AND 16#2000) <> 0) THEN
				iErrornumber			:=stParameterBuffer.iParameterReadValue[iBufferNumber];
				iParameterStep		:=5;
			ELSE
				iParameterReadvalue	:=stParameterBuffer.iParameterReadValue[iBufferNumber];
				iParameterStep		:=10;
			END_IF
			stParameterBuffer.iParameterStatus[iBufferNumber]	:=0;
			stParameterBuffer.iParameterReadValue[iBufferNumber]:=0;
		ELSIF TimerBuffer.Q THEN
			TimerBuffer(in:=FALSE);
			iErrornumber			:=1;
			iParameterStep		:=5;
		END_IF

		(*Errorstate*)
	5:	bErr				:=TRUE;
		bBusy			:=FALSE;
		bStart			:=FALSE;
		iParameterStep	:=10;

		(*Quit*)
	10:	IF (NOT bCycleMode) OR (NOT bStart) OR bErr THEN
			bBusy				:=FALSE;
			bStart				:=FALSE;
		END_IF
		iParameterStep	:=0;


	ELSE
		;
	END_CASE
END_FUNCTION_BLOCK

(* POU FB_ASI_ParameterControl, ST *)
(*********************************************************************************************************

NAME..............	:	FB_ParameterControl
DATE...............	:	21.04.2002
AUTHOR........	:	G.Sieder (Beckhoff Industrieelektronik)

DESCRIPTION:	internal FB to realize a multi-instance mode

		***	A CYCLIC CALLING OF THIS FB MUST BE GUARANTEED	***

HISTORY:	
21.03.2002	gs	start coding

*********************************************************************************************************)
FUNCTION_BLOCK FB_ASI_ParameterControl
VAR_INPUT
END_VAR
VAR_OUTPUT
END_VAR
VAR_IN_OUT
	stParameter_IN		:ST_Parameter_IN;
	stParameter_OUT		:ST_Parameter_OUT;
	stParameterBuffer		:ST_ParameterBuffer;
END_VAR
VAR
	bstatemashine		:BOOL;
	iBuffercounter			:INT;
	iBufferstate			:INT;
	bcheck				:BOOL;
	iParameterstate_old	:WORD;
	iBuffercounterOld		:INT;

END_VAR
	IF (NOT bstatemashine) THEN
		FOR iBuffercounter	:=0 TO 50 DO
			IF stParameterBuffer.ParameterControl[iBuffercounter] <> 0 THEN
				IF iBuffercounter >iBuffercounterOld OR iBuffercounterOld=50 THEN
					iBufferstate	:=1;
					EXIT;
				END_IF
			END_IF
		END_FOR
	END_IF

	CASE iBufferstate OF

	1:	bstatemashine	:=TRUE;
		(*check value of ToggleBit*)
		IF (stParameter_IN.iParameterStatus AND 2#0001000000000000)<>0 THEN
			bcheck	:=TRUE;
		ELSE
			bcheck	:=FALSE;
		END_IF
		iBufferstate		:=2;

	(*send Parameter to ASI-Master*)
	2:	IF iParameterstate_old = stParameterBuffer.ParameterControl[iBuffercounter] THEN
			stParameter_OUT.ParameterControl	:=stParameterBuffer.ParameterControl[iBuffercounter]+ 16#4000;
			stParameter_OUT.iParametervalue	:=stParameterBuffer.iParametervalue[iBuffercounter];
		ELSE
			stParameter_OUT.ParameterControl	:=stParameterBuffer.ParameterControl[iBuffercounter];
			stParameter_OUT.iParametervalue	:=stParameterBuffer.iParametervalue[iBuffercounter];
		END_IF
		iBufferstate	:=3;

	(*Read Parameter*)
	3:	IF (bcheck AND (stParameter_IN.iParameterStatus AND   2#0001000000000000) =0)
		OR (NOT bcheck AND (stParameter_IN.iParameterStatus AND 2#0001000000000000) <>0) THEN
			IF iParameterstate_old <> stParameter_OUT.ParameterControl  THEN
			(*IF iParameterstate_old <> stParameterBuffer.ParameterControl[iBuffercounter]  THEN*)
				stParameterBuffer.iParameterStatus[iBuffercounter]		:=stParameter_IN.iParameterStatus;
				stParameterBuffer.iParameterReadValue[iBuffercounter]	:=stParameter_IN.iParameterReadValue;
				stParameterBuffer.ParameterControl[iBuffercounter]		:=0;
				stParameterBuffer.iParametervalue[iBuffercounter]		:=0;
			ELSE
				stParameterBuffer.iParameterStatus[iBuffercounter]		:=0;
				stParameterBuffer.iParameterReadValue[iBuffercounter]	:=0;
			END_IF
			iParameterstate_old	:= stParameter_OUT.ParameterControl;
			iBufferstate			:=10;
		END_IF

	(*Quit*)
	10:	bstatemashine	:=FALSE;
		iBufferstate		:=0;
		iBuffercounterOld	:=iBuffercounter;
	ELSE
		;
	END_CASE
END_FUNCTION_BLOCK

(* POU FB_ASI_Processdata_analog, ST *)
(*********************************************************************************************************

NAME..............	:	FB_Processdata_analog
DATE...............	:	21.03.2002
AUTHOR........	:	G.Sieder (Beckhoff Industrieelektronik)

DESCRIPTION:	FB for Read/Write analog data from/to one Slave

HISTORY:	
21.03.2002	gs	start coding

*********************************************************************************************************)
FUNCTION_BLOCK FB_ASI_Processdata_analog
VAR_INPUT
	iSlaveaddress		:BYTE;
	iSlavevalue			:WORD;
	bParametermode		:BOOL;		(*0: Read, 1: Write *)
	bCycleMode			:BOOL;		(*0: Cyclic (permanent Read/Write), 1: Acyclic *)
	bCommMode			:BOOL;		(*0: Parameterzugriff, 1: ADS*)
	bRegComm			:BOOL;		(*Registerkommunikation: 0: Parameterzugriff, 1: Registerkommunikation *)
	bmaskAccess		:BOOL;		(*0:usual access, 1:mask access*)
	bStart				:BOOL;
END_VAR
VAR_OUTPUT
	bBusy				:BOOL;
	bErr					:BOOL;
	iErrornumber			:DWORD;
	iReadValue			:WORD;
	iParametergroup		:WORD;
END_VAR
VAR_IN_OUT
	stParameterBuffer		:ST_ParameterBuffer;
END_VAR
VAR
	fbParameterinterface	:FB_ASI_Parameterinterface;
	TrigStart				:R_TRIG;
	iParametermask		:WORD;
	bHiWord				:BOOL;
	iParametervalue		:DWORD;
	iParameterReadValue	:DWORD;
	istate				:INT;
END_VAR
	CASE istate OF

		0:	TrigStart(clk:=bStart);
			IF TrigStart.Q THEN
				bBusy		:=TRUE;
				bErr			:=FALSE;
				iErrornumber	:=0;
				istate		:=1;
			END_IF

		(*prepare Parametervalue*)
		1:	iParametervalue	:=0;
			iParametergroup	:=(iSlaveaddress-1)/2;
			iParametervalue	:=SHL((iParametervalue+iSlavevalue),(((iSlaveaddress-(iParametergroup*2))-1)*16));
			IF bmaskAccess THEN
				IF (iSlaveaddress- iParametergroup*2)> 4 THEN
					iParametermask	:=DWORD_TO_WORD(ROL(iParametervalue,16));
					bHiWord			:=TRUE;
				ELSE
					iParametermask	:=DWORD_TO_WORD(iParametervalue);
				END_IF
			END_IF
			istate	:=2;

		(*write Parametervalue*)
		2:	fbParameterinterface(iParameternumber	:=iParametergroup+16#90,
							iParametervalue		:=iParametervalue,
							stParameterBuffer		:=stParameterBuffer,
							bHiWord				:=bHiWord,
							bmaskAccess		:=bmaskAccess,
							iParametermask		:=iParametermask,
							bParametermode		:=bParametermode,
							bCycleMode			:=bCycleMode,
							bCommMode			:=bCommMode,
							bRegComm			:=bRegComm,
							bStart				:=TRUE);
			IF (NOT fbParameterinterface.bBusy) OR (NOT bCycleMode) THEN
				IF fbParameterinterface.bErr THEN
					bErr			:=TRUE;
					iErrornumber	:=fbParameterinterface.iErrornumber;
					istate	:=10;
				ELSIF (NOT bParametermode) OR (NOT bCycleMode) THEN
					iParameterReadValue	:=fbParameterinterface.iParameterReadvalue;
					istate	:=3;
				ELSE
					istate	:=3;
				END_IF
			END_IF

		(*read Parametervalue*)
		3:	iReadValue	:=DWORD_TO_WORD(SHR(iParameterReadValue,((iSlaveaddress-(iParametergroup*2))-1)*16));
			IF (NOT bStart) OR ( bCycleMode) THEN
				fbParameterinterface(bStart			:=FALSE,
								stParameterBuffer	:=stParameterBuffer);
				IF (NOT fbParameterinterface.bBusy) THEN
					istate	:=10;
				END_IF
			ELSE
				istate	:=2;
			END_IF

			(*Quit*)
		10:	bBusy	:=FALSE;
			IF (NOT bStart) THEN
				istate	:=0;
			END_IF

	ELSE
		;
	END_CASE
END_FUNCTION_BLOCK

(* POU FB_ASI_Processdata_digital, ST *)
(*********************************************************************************************************

NAME..............	:	FB_Processdata_digital
DATE...............	:	21.03.2002
AUTHOR........	:	G.Sieder (Beckhoff Industrieelektronik)

DESCRIPTION:	FB for Read/Write digital data from/to one Slave

HISTORY:	
21.03.2002	gs	start coding

*********************************************************************************************************)
FUNCTION_BLOCK FB_ASI_Processdata_digital
VAR_INPUT
	iSlaveaddress		:BYTE;
	iSlavevalue			:BYTE;
	bParametermode		:BOOL;		(*0: Read, 1: Write *)
	bCycleMode			:BOOL;		(*0: Acyclic , 1:Cyclic (permanent Read/Write) *)
	bCommMode			:BOOL;		(*0: Parameterzugriff, 1: ADS*)
	bRegComm			:BOOL;		(*Registerkommunikation: 0: Parameterzugriff, 1: Registerkommunikation *)
	bmaskAccess		:BOOL;		(*0:usual access, 1:mask access*)
	bStart				:BOOL;
END_VAR
VAR_OUTPUT
	bBusy				:BOOL;
	bErr					:BOOL;
	iErrornumber			:DWORD;
	iReadValue			:BYTE;
	iParametergroup		:WORD;
END_VAR
VAR_IN_OUT
	stParameterBuffer		:ST_ParameterBuffer;
END_VAR
VAR
	fbParameterinterface	:FB_ASI_Parameterinterface;
	TrigStart				:R_TRIG;
	iParametermask		:WORD;
	bHiWord				:BOOL;
	iParametervalue		:DWORD;
	iParameterReadValue	:DWORD;
	istate				:INT;
END_VAR
	CASE istate OF

		0:	TrigStart(clk:=bStart);
			IF TrigStart.Q THEN
				bBusy		:=TRUE;
				bErr			:=FALSE;
				iErrornumber	:=0;
				istate		:=1;
			END_IF

		(*prepare Parametervalue*)
		1:	iParametervalue	:=0;
			iParametergroup	:=iSlaveaddress/8;
			(*iParametervalue	:=SHL((iParametervalue+iSlavevalue),(((iSlaveaddress-(iParametergroup*8))-1)*4));*)
			IF bmaskAccess THEN
				IF (iSlaveaddress- iParametergroup*8)> 4 THEN
					iParametermask	:=DWORD_TO_WORD(ROL(iParametervalue,16));
					bHiWord			:=TRUE;
				ELSE
					iParametermask	:=DWORD_TO_WORD(iParametervalue);
				END_IF
			END_IF
			istate	:=2;

		(*write Parametervalue*)
		2:	fbParameterinterface(iParameternumber	:=iSlaveaddress/8+16#80,
							iParametervalue		:=iParametervalue,
							stParameterBuffer		:=stParameterBuffer,
							bHiWord				:=bHiWord,
							bmaskAccess		:=bmaskAccess,
							iParametermask		:=iParametermask,
							bParametermode		:=bParametermode,
							bCycleMode			:=bCycleMode,
							bCommMode			:=bCommMode,
							bRegComm			:=bRegComm,
							bStart				:=TRUE);
			IF (NOT fbParameterinterface.bBusy) OR bCycleMode THEN
				IF fbParameterinterface.bErr THEN
					bErr			:=TRUE;
					iErrornumber	:=fbParameterinterface.iErrornumber;
					fbParameterinterface(bStart			:=FALSE,
									stParameterBuffer	:=stParameterBuffer);
					istate	:=10;
				ELSIF (NOT bParametermode) OR bCycleMode THEN
					iParameterReadValue	:=fbParameterinterface.iParameterReadvalue;
					istate	:=3;
				ELSE
					istate	:=3;
				END_IF
			END_IF

		(*read Parametervalue*)
		3:	iReadValue	:=(DWORD_TO_BYTE(SHR(iParameterReadValue,((iSlaveaddress-(iParametergroup*8))*4)))) AND 2#00001111;
			IF (NOT bStart) OR ( NOT bCycleMode) THEN
				fbParameterinterface(bStart			:=FALSE,
								stParameterBuffer	:=stParameterBuffer);
				IF (NOT fbParameterinterface.bBusy) THEN
					istate	:=10;
				END_IF
			ELSE
				istate	:=2;
			END_IF

			(*Quit*)
		10:	bBusy	:=FALSE;
			IF (NOT bStart) THEN
				istate	:=0;
			END_IF

	ELSE
		;
	END_CASE
END_FUNCTION_BLOCK

(* POU FB_ASI_Projecting, ST *)
(*********************************************************************************************************

NAME..............	:	FB_Projecting
DATE...............	:	21.03.2002
AUTHOR........	:	G.Sieder (Beckhoff Industrieelektronik)

DESCRIPTION:	FB to Read/Write Parameters for the slave-configuration 

HISTORY:	
21.03.2002	gs	start coding

*********************************************************************************************************)
FUNCTION_BLOCK FB_ASI_Projecting
VAR_INPUT
	iSlaveaddress		:BYTE;
	iParametervalue		:DWORD;
	bIOValue			:BOOL;	(*Read/Write IO-value of a slave*)
	bIDCode				:BOOL;	(*Read/Write	ID-code of a slave*)
	bReadWrite			:BOOL;	(*0: Read, 1: Write*)
	bReadLPS			:BOOL;	(*Read List of all projected Slaves*)
	bStart				:BOOL;
END_VAR
VAR_OUTPUT
	bBusy				:BOOL;
	bErr					:BOOL;
	iErrornumber			:DWORD;
	iParameterReadvalue	:BYTE;	(*IO-value or ID-code of a slave*)
	iLPS				:DWORD;
END_VAR
VAR_IN_OUT
	stParameterBuffer		:ST_ParameterBuffer;
END_VAR
VAR
	iProjectingStep	:INT;
	TrigStart			:R_TRIG;
	iAddressFactor	:BYTE;
	iParameternumber	:WORD;
	iReadValue		:DWORD;
	fbParameterinterface	:FB_ASI_Parameterinterface;
END_VAR
	CASE iProjectingStep OF

	(*Idle*)
	0:	TrigStart(clk:=bStart);
		IF TrigStart.Q THEN
			bBusy				:=TRUE;
			bErr					:=FALSE;
			iErrornumber			:=0;
			iProjectingStep		:=1;
		END_IF

